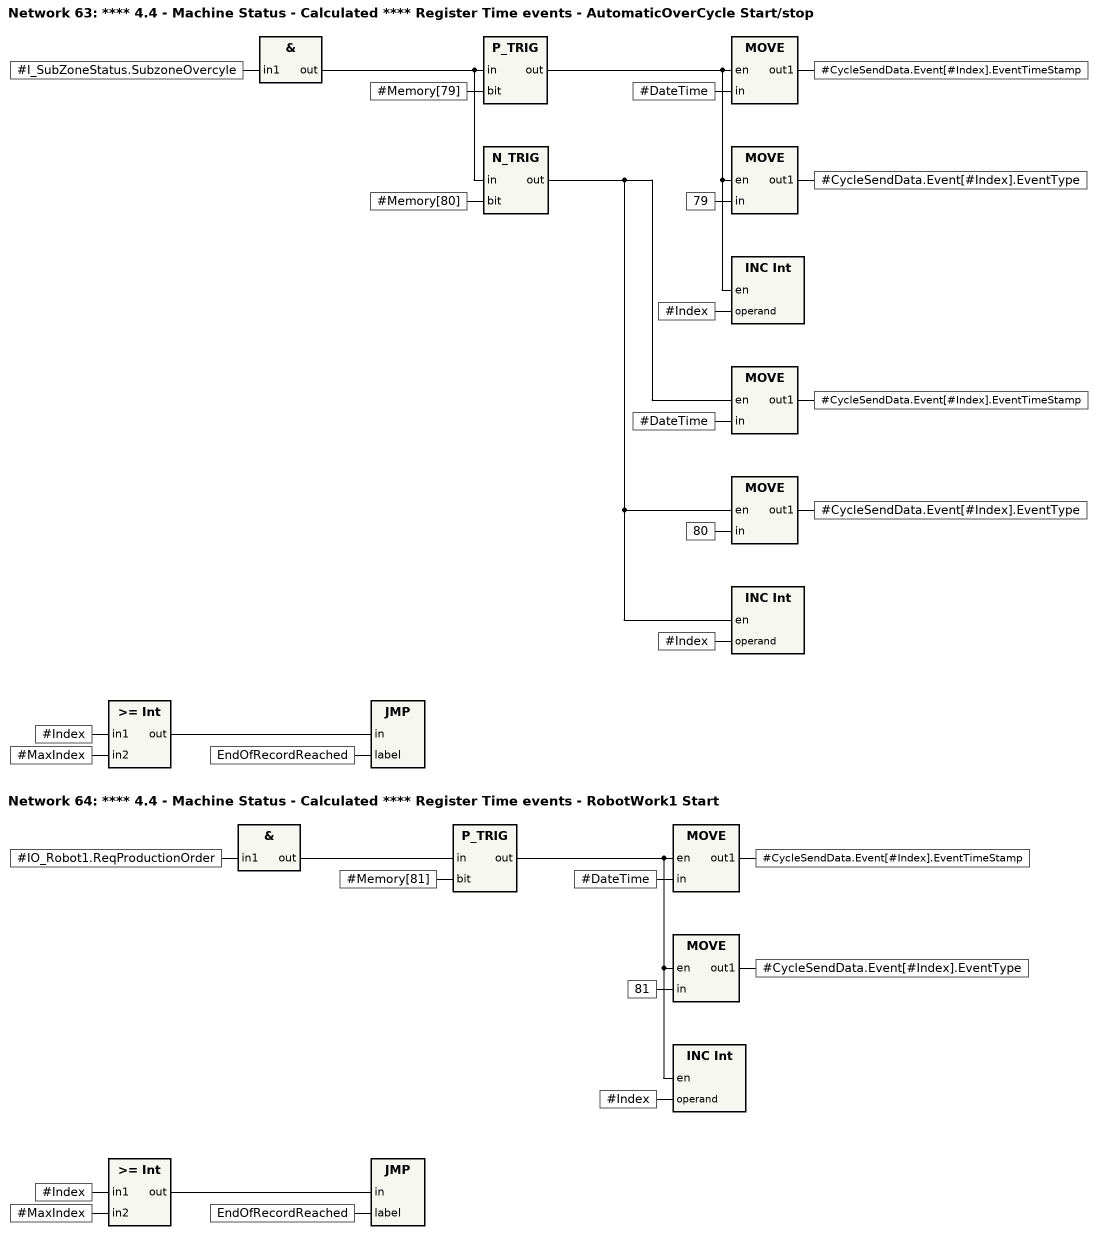
   #_w1 := #I_SubZoneStatus.SubzoneOvercyle AND NOT #Memory[79];   // rising edge
   #Memory[79] := #I_SubZoneStatus.SubzoneOvercyle;
   IF #_w1 THEN
       #CycleSendData.Event[#Index].EventTimeStamp := #DateTime;
       #CycleSendData.Event[#Index].EventType := 79;
       #Index := #Index + 1;
   END_IF;
   #_w2 := NOT #I_SubZoneStatus.SubzoneOvercyle AND #Memory[80];   // falling edge
   #Memory[80] := #I_SubZoneStatus.SubzoneOvercyle;
   IF #_w2 THEN
       #CycleSendData.Event[#Index].EventTimeStamp := #DateTime;
       #CycleSendData.Event[#Index].EventType := 80;
       #Index := #Index + 1;
   END_IF;
   IF #Index >= #MaxIndex THEN GOTO EndOfRecordReached; END_IF;
END_REGION

REGION Network 64: **** 4.4 - Machine Status - Calculated **** Register Time events - RobotWork1 Start
   #_w1 := #IO_Robot1.ReqProductionOrder AND NOT #Memory[81];   // rising edge
   #Memory[81] := #IO_Robot1.ReqProductionOrder;
   IF #_w1 THEN
       #CycleSendData.Event[#Index].EventTimeStamp := #DateTime;
       #CycleSendData.Event[#Index].EventType := 81;
       #Index := #Index + 1;
   END_IF;
   IF #Index >= #MaxIndex THEN GOTO EndOfRecordReached; END_IF;
END_REGION

REGION Network 65: **** 4.4 - Machine Status - Calculated **** Register Time events - RobotWork1 Stop
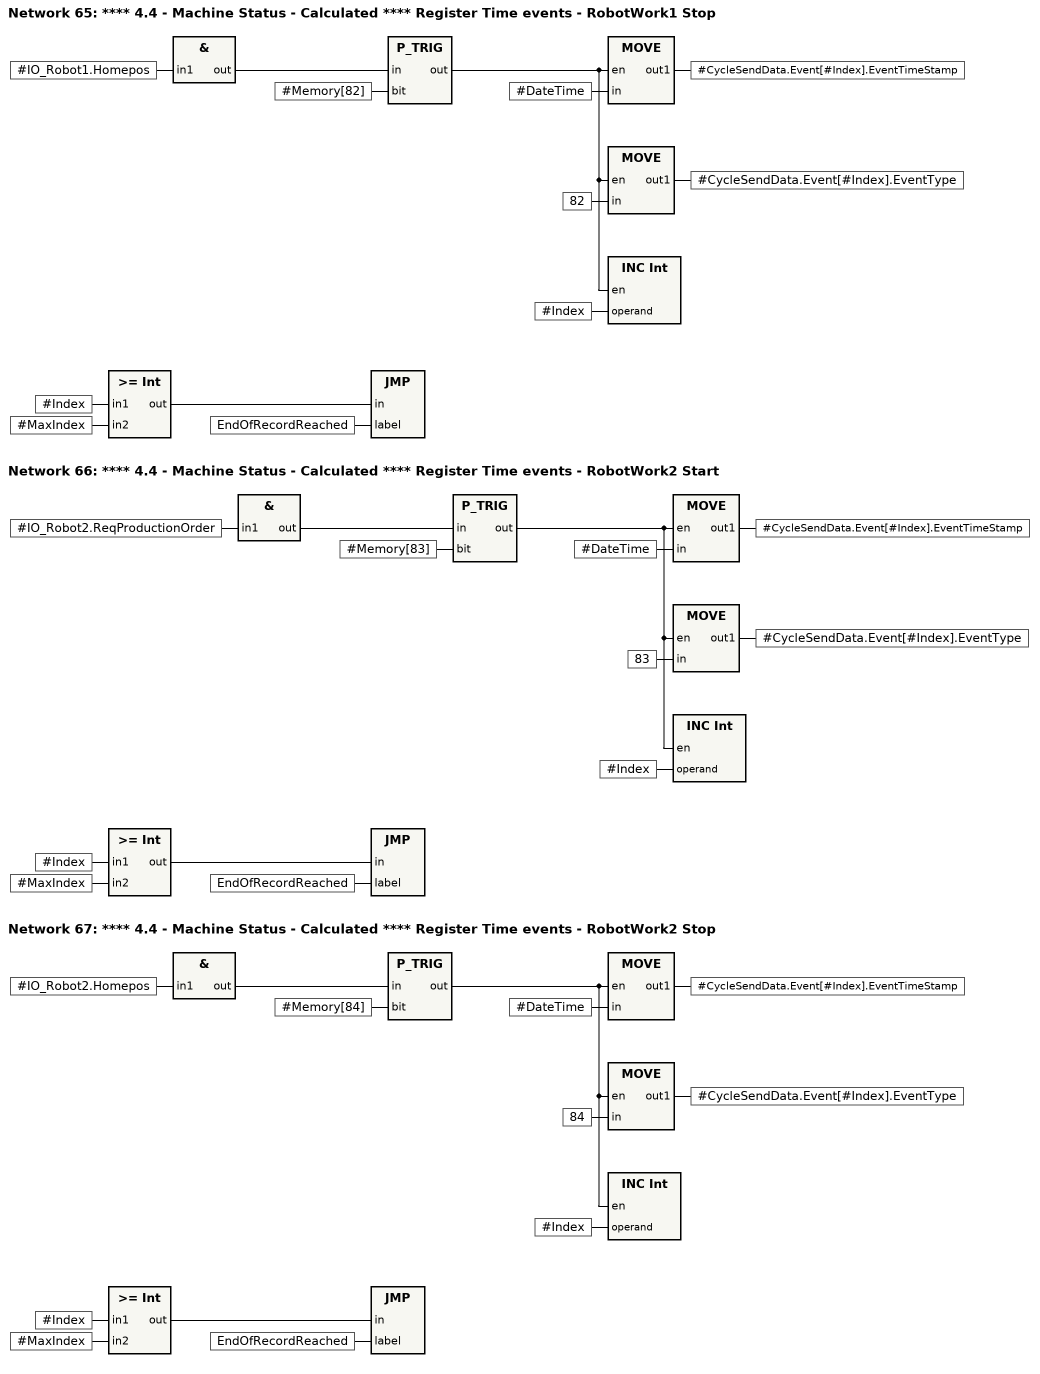
   #_w1 := #IO_Robot1.Homepos AND NOT #Memory[82];   // rising edge
   #Memory[82] := #IO_Robot1.Homepos;
   IF #_w1 THEN
       #CycleSendData.Event[#Index].EventTimeStamp := #DateTime;
       #CycleSendData.Event[#Index].EventType := 82;
       #Index := #Index + 1;
   END_IF;
   IF #Index >= #MaxIndex THEN GOTO EndOfRecordReached; END_IF;
END_REGION

REGION Network 66: **** 4.4 - Machine Status - Calculated **** Register Time events - RobotWork2 Start
   #_w1 := #IO_Robot2.ReqProductionOrder AND NOT #Memory[83];   // rising edge
   #Memory[83] := #IO_Robot2.ReqProductionOrder;
   IF #_w1 THEN
       #CycleSendData.Event[#Index].EventTimeStamp := #DateTime;
       #CycleSendData.Event[#Index].EventType := 83;
       #Index := #Index + 1;
   END_IF;
   IF #Index >= #MaxIndex THEN GOTO EndOfRecordReached; END_IF;
END_REGION

REGION Network 67: **** 4.4 - Machine Status - Calculated **** Register Time events - RobotWork2 Stop
   #_w1 := #IO_Robot2.Homepos AND NOT #Memory[84];   // rising edge
   #Memory[84] := #IO_Robot2.Homepos;
   IF #_w1 THEN
       #CycleSendData.Event[#Index].EventTimeStamp := #DateTime;
       #CycleSendData.Event[#Index].EventType := 84;
       #Index := #Index + 1;
   END_IF;
   IF #Index >= #MaxIndex THEN GOTO EndOfRecordReached; END_IF;
END_REGION

REGION Network 68: **** 4.4 - Machine Status - Calculated **** Register Time events - RobotWork3 Start
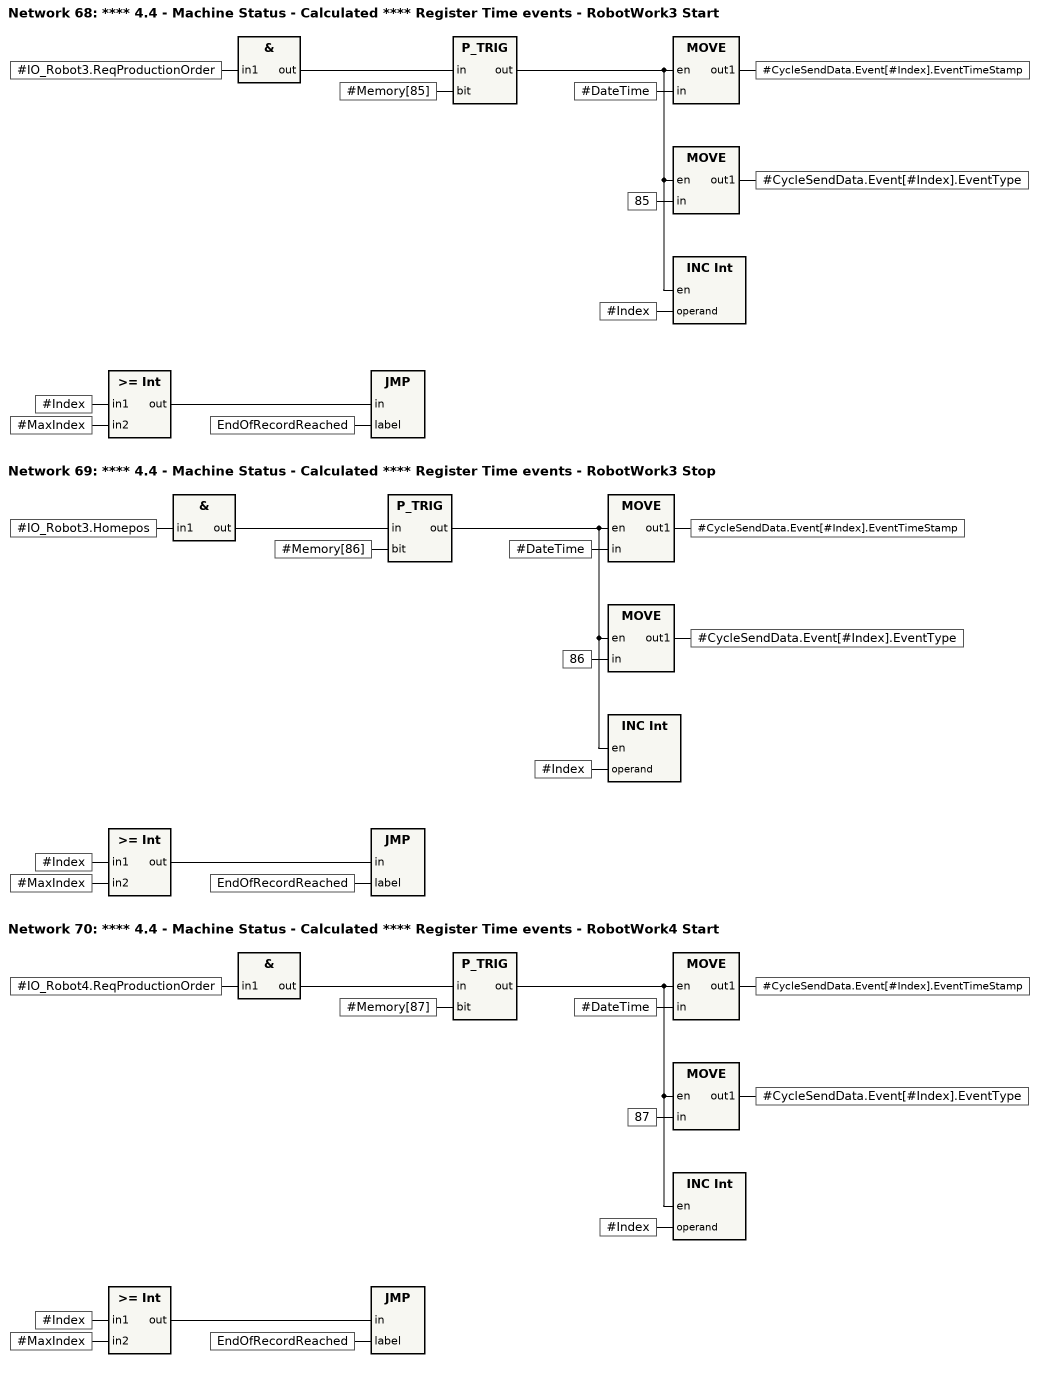
   #_w1 := #IO_Robot3.ReqProductionOrder AND NOT #Memory[85];   // rising edge
   #Memory[85] := #IO_Robot3.ReqProductionOrder;
   IF #_w1 THEN
       #CycleSendData.Event[#Index].EventTimeStamp := #DateTime;
       #CycleSendData.Event[#Index].EventType := 85;
       #Index := #Index + 1;
   END_IF;
   IF #Index >= #MaxIndex THEN GOTO EndOfRecordReached; END_IF;
END_REGION

REGION Network 69: **** 4.4 - Machine Status - Calculated **** Register Time events - RobotWork3 Stop
   #_w1 := #IO_Robot3.Homepos AND NOT #Memory[86];   // rising edge
   #Memory[86] := #IO_Robot3.Homepos;
   IF #_w1 THEN
       #CycleSendData.Event[#Index].EventTimeStamp := #DateTime;
       #CycleSendData.Event[#Index].EventType := 86;
       #Index := #Index + 1;
   END_IF;
   IF #Index >= #MaxIndex THEN GOTO EndOfRecordReached; END_IF;
END_REGION

REGION Network 70: **** 4.4 - Machine Status - Calculated **** Register Time events - RobotWork4 Start
   #_w1 := #IO_Robot4.ReqProductionOrder AND NOT #Memory[87];   // rising edge
   #Memory[87] := #IO_Robot4.ReqProductionOrder;
   IF #_w1 THEN
       #CycleSendData.Event[#Index].EventTimeStamp := #DateTime;
       #CycleSendData.Event[#Index].EventType := 87;
       #Index := #Index + 1;
   END_IF;
   IF #Index >= #MaxIndex THEN GOTO EndOfRecordReached; END_IF;
END_REGION

REGION Network 71: **** 4.4 - Machine Status - Calculated **** Register Time events - RobotWork4 Stop
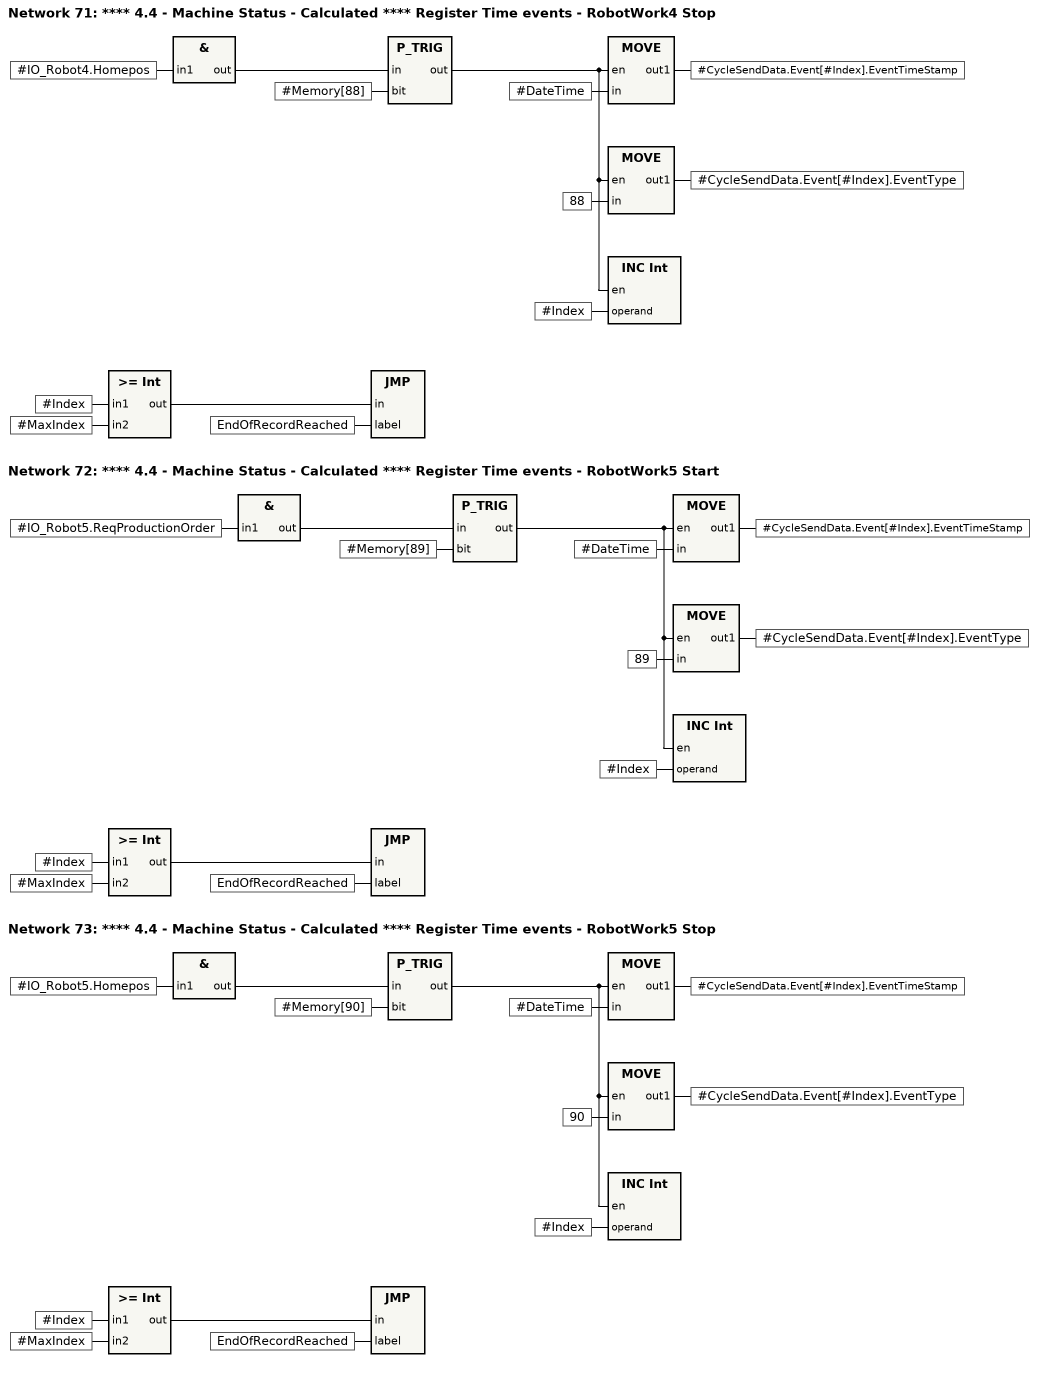
   #_w1 := #IO_Robot4.Homepos AND NOT #Memory[88];   // rising edge
   #Memory[88] := #IO_Robot4.Homepos;
   IF #_w1 THEN
       #CycleSendData.Event[#Index].EventTimeStamp := #DateTime;
       #CycleSendData.Event[#Index].EventType := 88;
       #Index := #Index + 1;
   END_IF;
   IF #Index >= #MaxIndex THEN GOTO EndOfRecordReached; END_IF;
END_REGION

REGION Network 72: **** 4.4 - Machine Status - Calculated **** Register Time events - RobotWork5 Start
   #_w1 := #IO_Robot5.ReqProductionOrder AND NOT #Memory[89];   // rising edge
   #Memory[89] := #IO_Robot5.ReqProductionOrder;
   IF #_w1 THEN
       #CycleSendData.Event[#Index].EventTimeStamp := #DateTime;
       #CycleSendData.Event[#Index].EventType := 89;
       #Index := #Index + 1;
   END_IF;
   IF #Index >= #MaxIndex THEN GOTO EndOfRecordReached; END_IF;
END_REGION

REGION Network 73: **** 4.4 - Machine Status - Calculated **** Register Time events - RobotWork5 Stop
   #_w1 := #IO_Robot5.Homepos AND NOT #Memory[90];   // rising edge
   #Memory[90] := #IO_Robot5.Homepos;
   IF #_w1 THEN
       #CycleSendData.Event[#Index].EventTimeStamp := #DateTime;
       #CycleSendData.Event[#Index].EventType := 90;
       #Index := #Index + 1;
   END_IF;
   IF #Index >= #MaxIndex THEN GOTO EndOfRecordReached; END_IF;
END_REGION

REGION Network 74: **** 4.4 - Machine Status - Calculated **** Register Time events - RobotWork6 Start
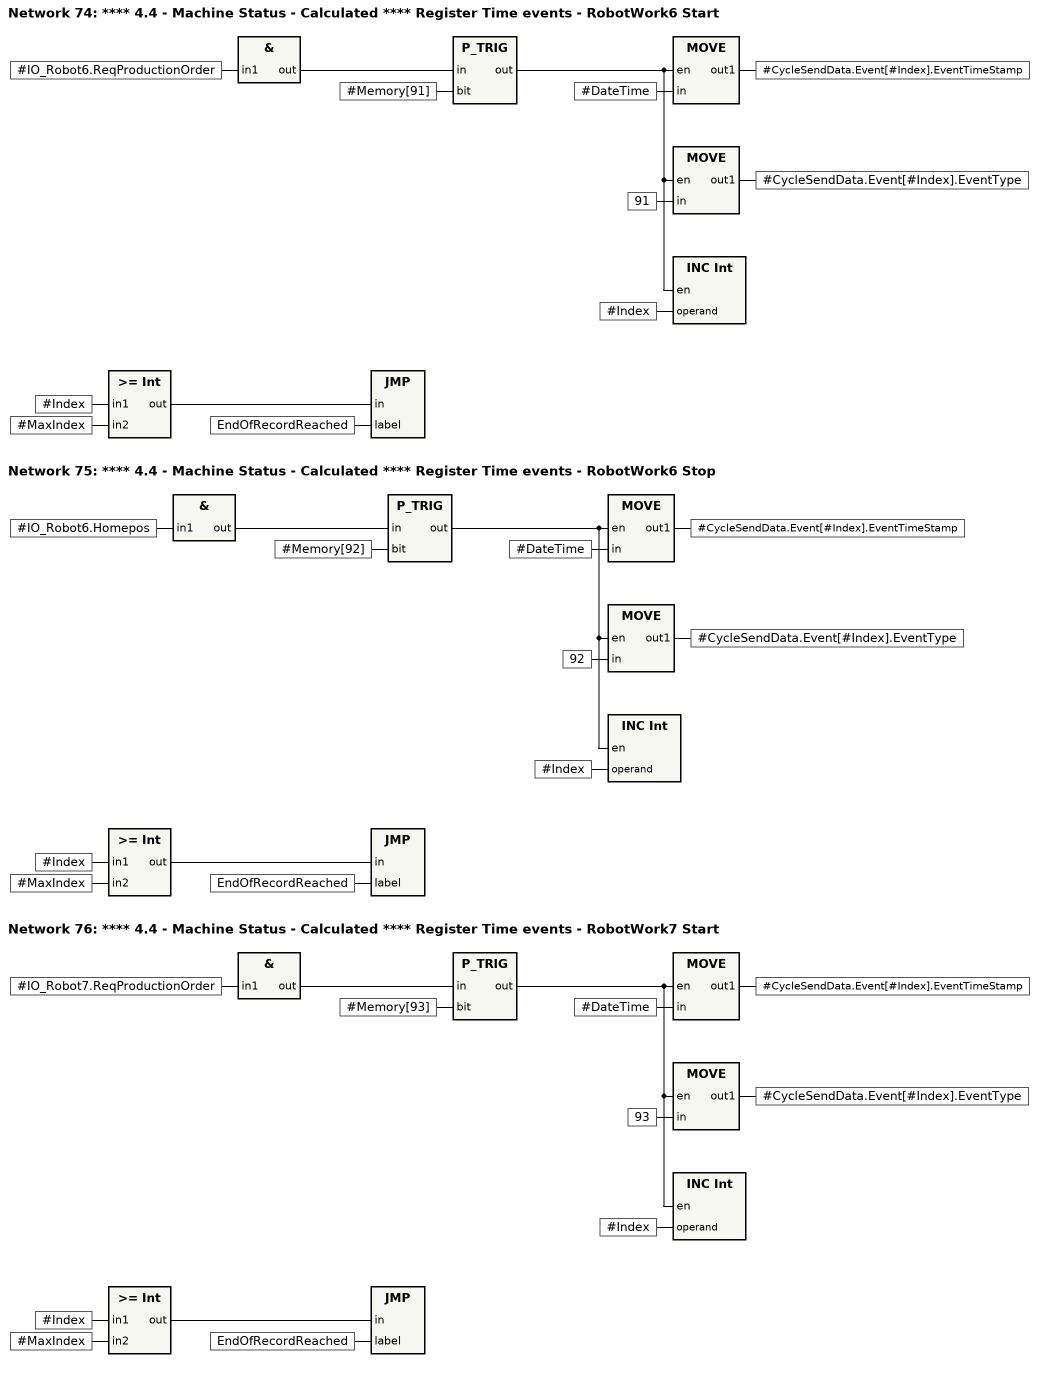
   #_w1 := #IO_Robot6.ReqProductionOrder AND NOT #Memory[91];   // rising edge
   #Memory[91] := #IO_Robot6.ReqProductionOrder;
   IF #_w1 THEN
       #CycleSendData.Event[#Index].EventTimeStamp := #DateTime;
       #CycleSendData.Event[#Index].EventType := 91;
       #Index := #Index + 1;
   END_IF;
   IF #Index >= #MaxIndex THEN GOTO EndOfRecordReached; END_IF;
END_REGION

REGION Network 75: **** 4.4 - Machine Status - Calculated **** Register Time events - RobotWork6 Stop
   #_w1 := #IO_Robot6.Homepos AND NOT #Memory[92];   // rising edge
   #Memory[92] := #IO_Robot6.Homepos;
   IF #_w1 THEN
       #CycleSendData.Event[#Index].EventTimeStamp := #DateTime;
       #CycleSendData.Event[#Index].EventType := 92;
       #Index := #Index + 1;
   END_IF;
   IF #Index >= #MaxIndex THEN GOTO EndOfRecordReached; END_IF;
END_REGION

REGION Network 76: **** 4.4 - Machine Status - Calculated **** Register Time events - RobotWork7 Start
   #_w1 := #IO_Robot7.ReqProductionOrder AND NOT #Memory[93];   // rising edge
   #Memory[93] := #IO_Robot7.ReqProductionOrder;
   IF #_w1 THEN
       #CycleSendData.Event[#Index].EventTimeStamp := #DateTime;
       #CycleSendData.Event[#Index].EventType := 93;
       #Index := #Index + 1;
   END_IF;
   IF #Index >= #MaxIndex THEN GOTO EndOfRecordReached; END_IF;
END_REGION

REGION Network 77: **** 4.4 - Machine Status - Calculated **** Register Time events - RobotWork7 Stop
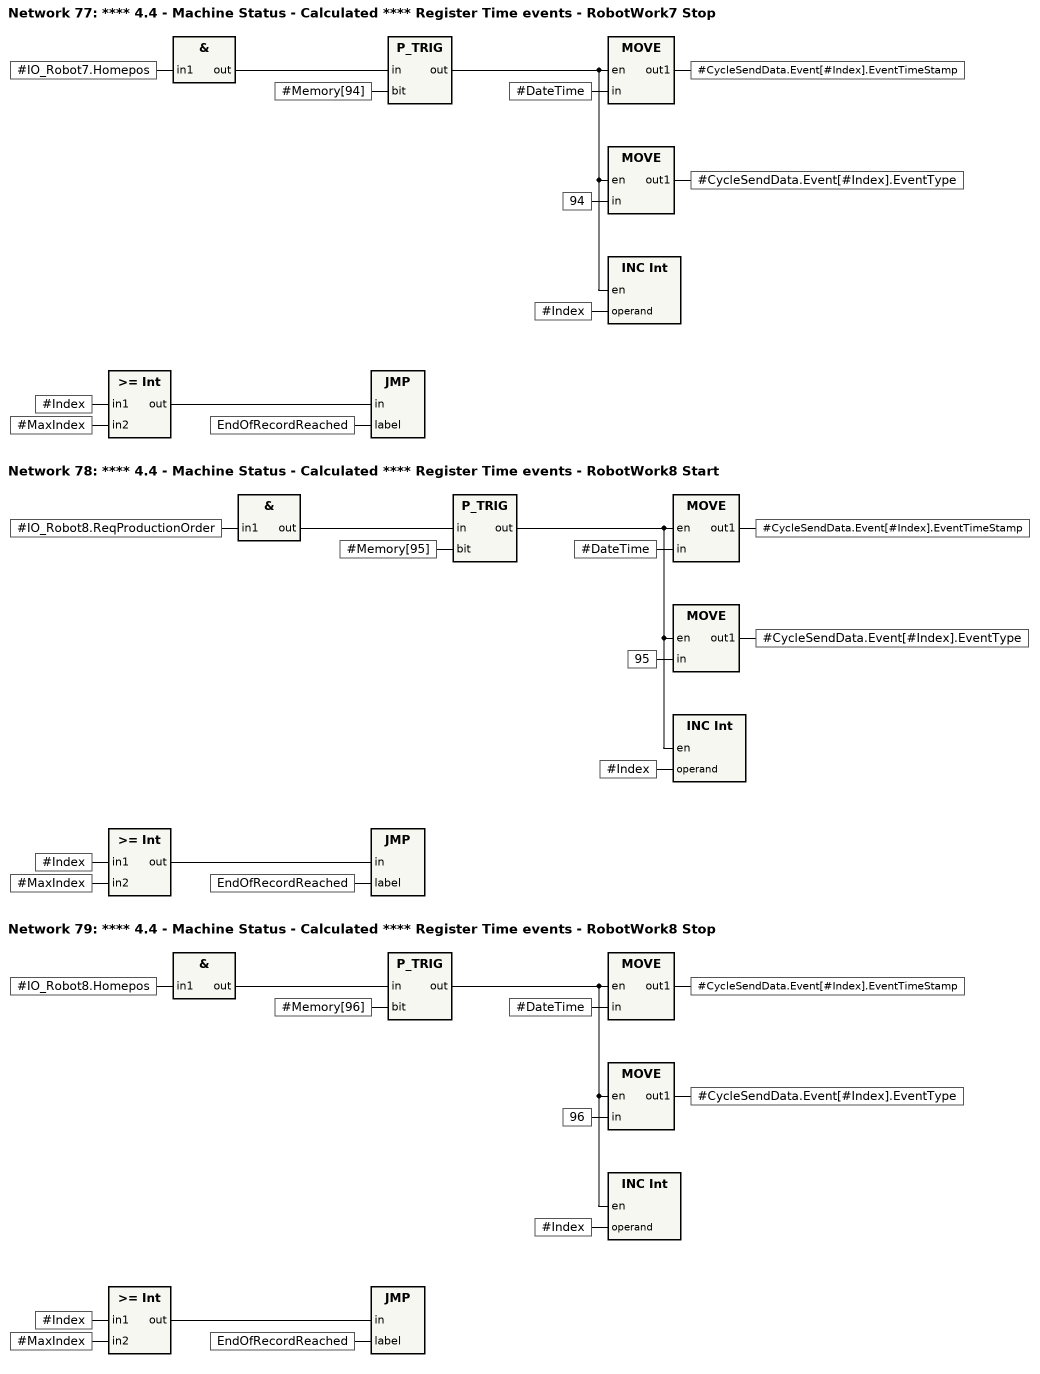
   #_w1 := #IO_Robot7.Homepos AND NOT #Memory[94];   // rising edge
   #Memory[94] := #IO_Robot7.Homepos;
   IF #_w1 THEN
       #CycleSendData.Event[#Index].EventTimeStamp := #DateTime;
       #CycleSendData.Event[#Index].EventType := 94;
       #Index := #Index + 1;
   END_IF;
   IF #Index >= #MaxIndex THEN GOTO EndOfRecordReached; END_IF;
END_REGION

REGION Network 78: **** 4.4 - Machine Status - Calculated **** Register Time events - RobotWork8 Start
   #_w1 := #IO_Robot8.ReqProductionOrder AND NOT #Memory[95];   // rising edge
   #Memory[95] := #IO_Robot8.ReqProductionOrder;
   IF #_w1 THEN
       #CycleSendData.Event[#Index].EventTimeStamp := #DateTime;
       #CycleSendData.Event[#Index].EventType := 95;
       #Index := #Index + 1;
   END_IF;
   IF #Index >= #MaxIndex THEN GOTO EndOfRecordReached; END_IF;
END_REGION

REGION Network 79: **** 4.4 - Machine Status - Calculated **** Register Time events - RobotWork8 Stop
   #_w1 := #IO_Robot8.Homepos AND NOT #Memory[96];   // rising edge
   #Memory[96] := #IO_Robot8.Homepos;
   IF #_w1 THEN
       #CycleSendData.Event[#Index].EventTimeStamp := #DateTime;
       #CycleSendData.Event[#Index].EventType := 96;
       #Index := #Index + 1;
   END_IF;
   IF #Index >= #MaxIndex THEN GOTO EndOfRecordReached; END_IF;
END_REGION

REGION Network 80: **** 4.4 - Machine Status - Calculated **** Register Time events - RobotWork9 Start
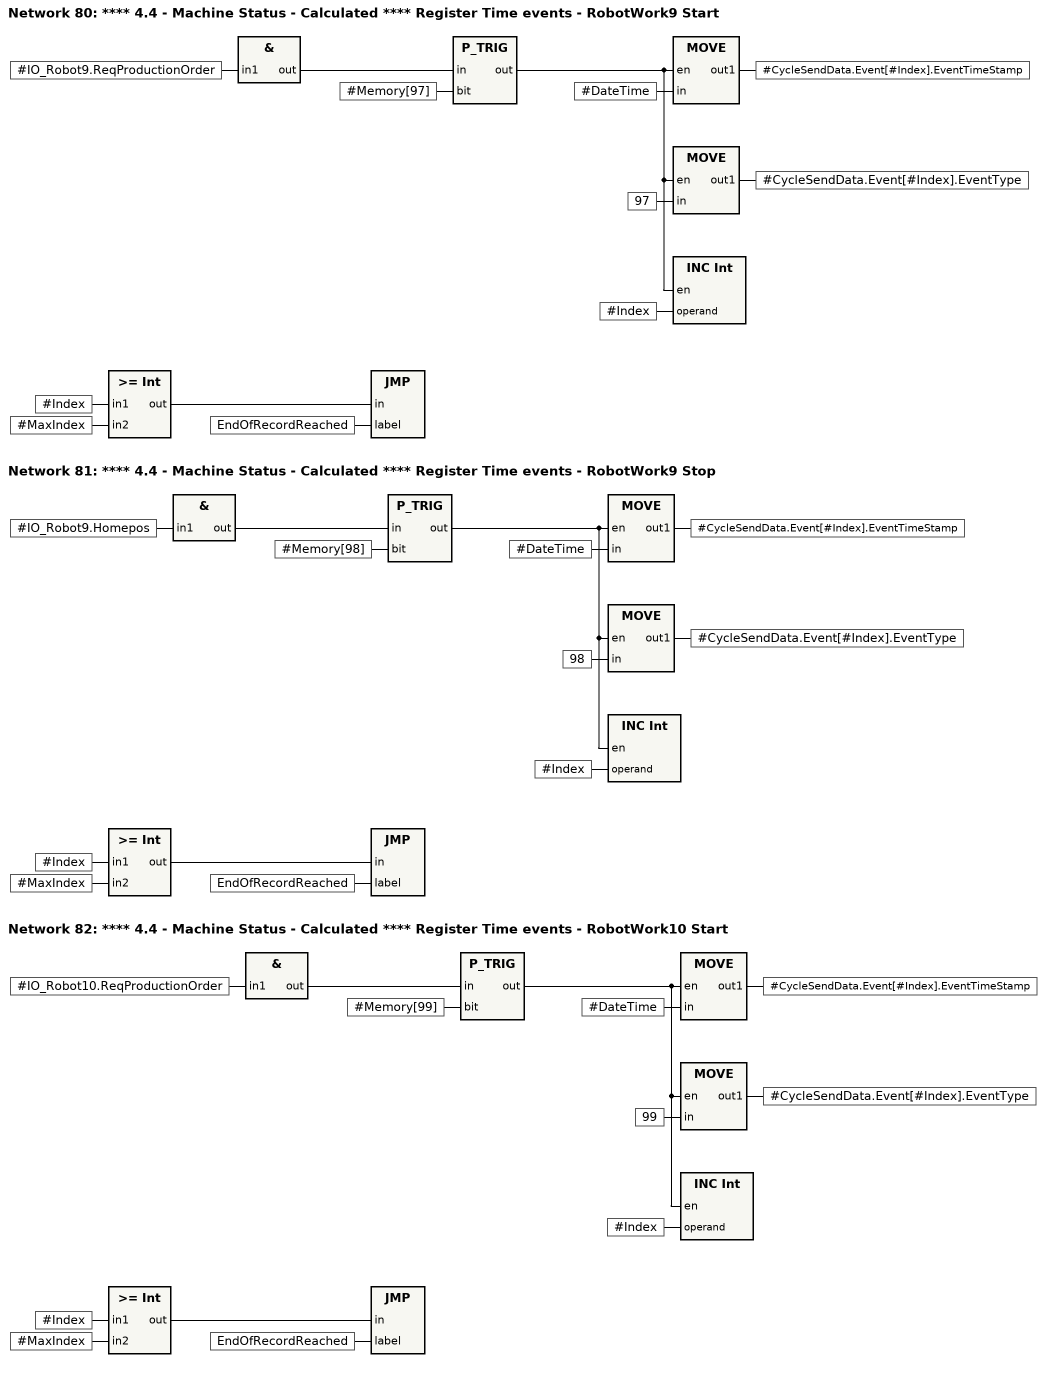
   #_w1 := #IO_Robot9.ReqProductionOrder AND NOT #Memory[97];   // rising edge
   #Memory[97] := #IO_Robot9.ReqProductionOrder;
   IF #_w1 THEN
       #CycleSendData.Event[#Index].EventTimeStamp := #DateTime;
       #CycleSendData.Event[#Index].EventType := 97;
       #Index := #Index + 1;
   END_IF;
   IF #Index >= #MaxIndex THEN GOTO EndOfRecordReached; END_IF;
END_REGION

REGION Network 81: **** 4.4 - Machine Status - Calculated **** Register Time events - RobotWork9 Stop
   #_w1 := #IO_Robot9.Homepos AND NOT #Memory[98];   // rising edge
   #Memory[98] := #IO_Robot9.Homepos;
   IF #_w1 THEN
       #CycleSendData.Event[#Index].EventTimeStamp := #DateTime;
       #CycleSendData.Event[#Index].EventType := 98;
       #Index := #Index + 1;
   END_IF;
   IF #Index >= #MaxIndex THEN GOTO EndOfRecordReached; END_IF;
END_REGION

REGION Network 82: **** 4.4 - Machine Status - Calculated **** Register Time events - RobotWork10 Start
   #_w1 := #IO_Robot10.ReqProductionOrder AND NOT #Memory[99];   // rising edge
   #Memory[99] := #IO_Robot10.ReqProductionOrder;
   IF #_w1 THEN
       #CycleSendData.Event[#Index].EventTimeStamp := #DateTime;
       #CycleSendData.Event[#Index].EventType := 99;
       #Index := #Index + 1;
   END_IF;
   IF #Index >= #MaxIndex THEN GOTO EndOfRecordReached; END_IF;
END_REGION

REGION Network 83: **** 4.4 - Machine Status - Calculated **** Register Time events - RobotWork10 Stop
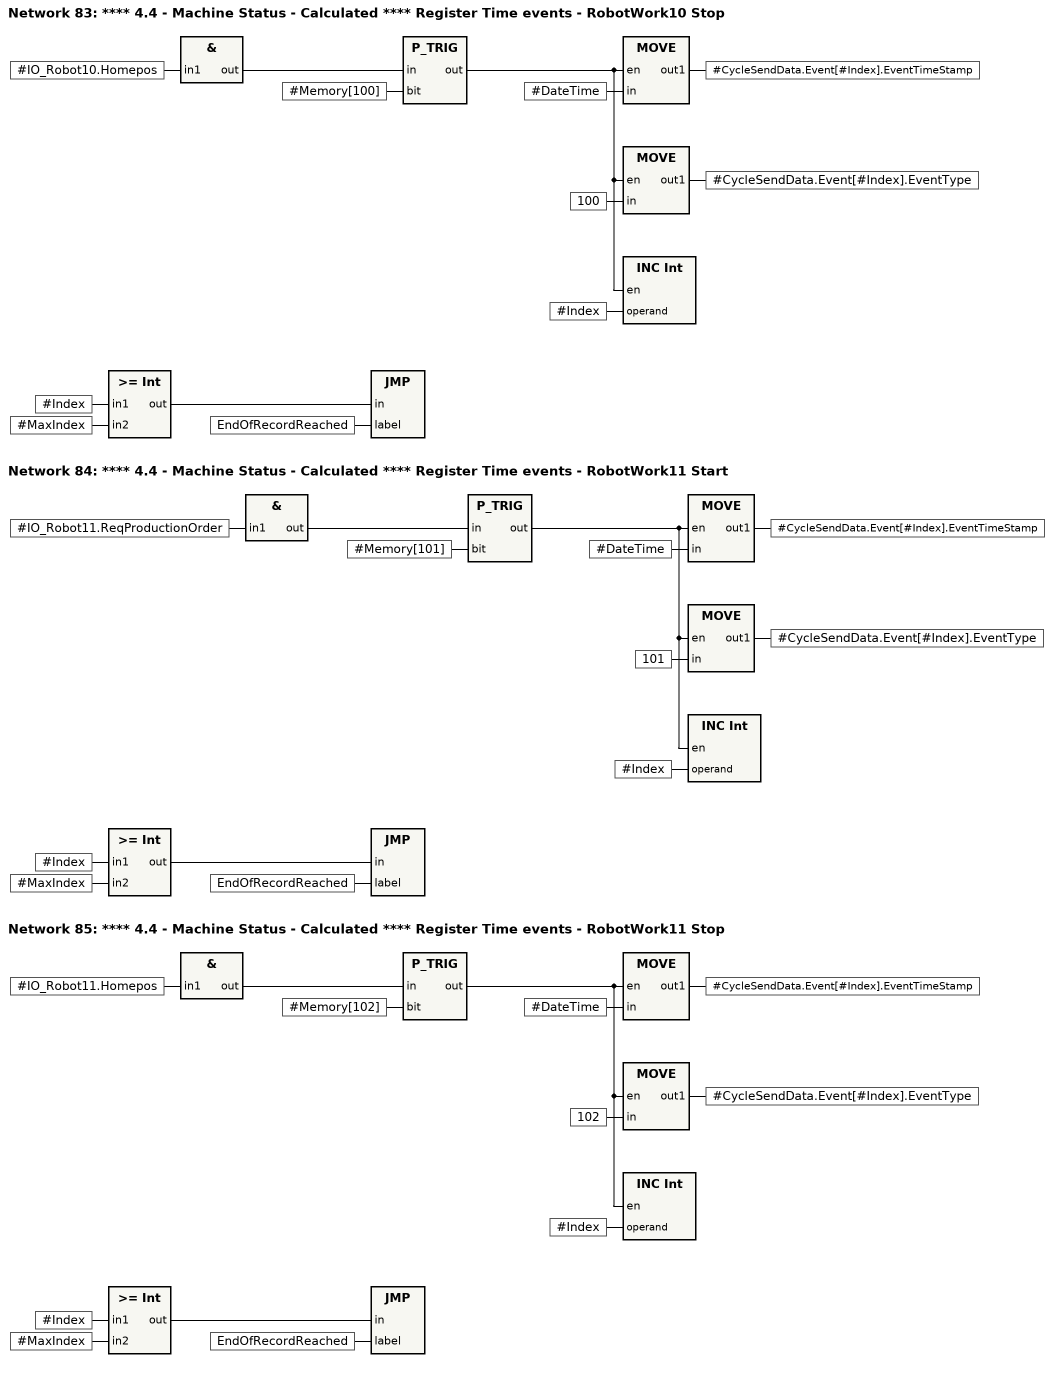
   #_w1 := #IO_Robot10.Homepos AND NOT #Memory[100];   // rising edge
   #Memory[100] := #IO_Robot10.Homepos;
   IF #_w1 THEN
       #CycleSendData.Event[#Index].EventTimeStamp := #DateTime;
       #CycleSendData.Event[#Index].EventType := 100;
       #Index := #Index + 1;
   END_IF;
   IF #Index >= #MaxIndex THEN GOTO EndOfRecordReached; END_IF;
END_REGION

REGION Network 84: **** 4.4 - Machine Status - Calculated **** Register Time events - RobotWork11 Start
   #_w1 := #IO_Robot11.ReqProductionOrder AND NOT #Memory[101];   // rising edge
   #Memory[101] := #IO_Robot11.ReqProductionOrder;
   IF #_w1 THEN
       #CycleSendData.Event[#Index].EventTimeStamp := #DateTime;
       #CycleSendData.Event[#Index].EventType := 101;
       #Index := #Index + 1;
   END_IF;
   IF #Index >= #MaxIndex THEN GOTO EndOfRecordReached; END_IF;
END_REGION

REGION Network 85: **** 4.4 - Machine Status - Calculated **** Register Time events - RobotWork11 Stop
   #_w1 := #IO_Robot11.Homepos AND NOT #Memory[102];   // rising edge
   #Memory[102] := #IO_Robot11.Homepos;
   IF #_w1 THEN
       #CycleSendData.Event[#Index].EventTimeStamp := #DateTime;
       #CycleSendData.Event[#Index].EventType := 102;
       #Index := #Index + 1;
   END_IF;
   IF #Index >= #MaxIndex THEN GOTO EndOfRecordReached; END_IF;
END_REGION

REGION Network 86: **** 4.4 - Machine Status - Calculated **** Register Time events - RobotWork12 Start
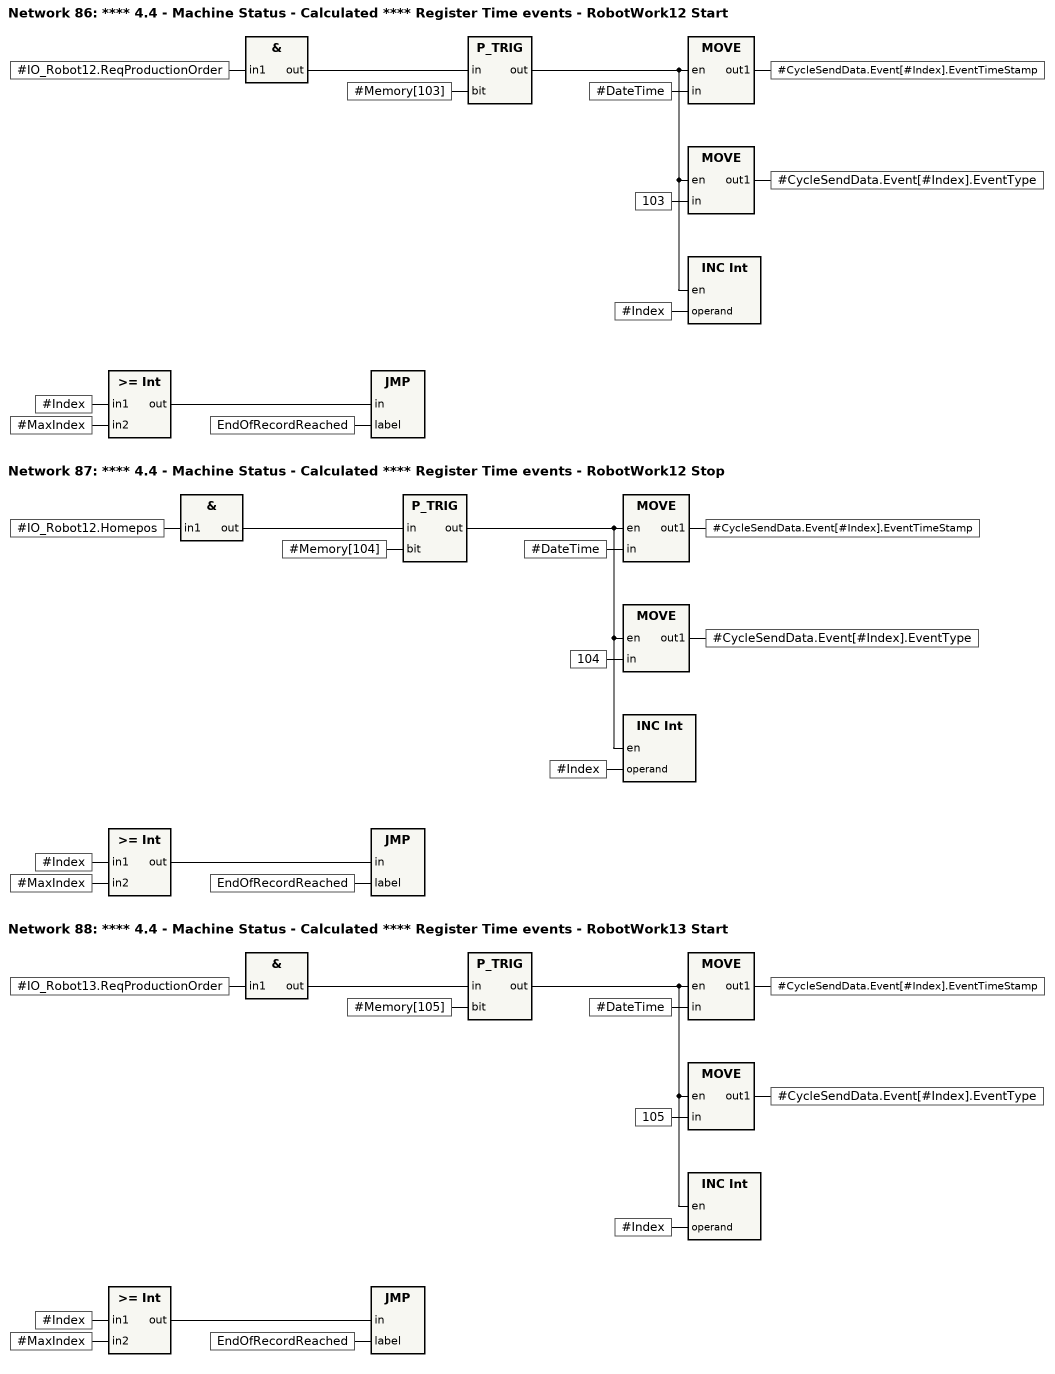
   #_w1 := #IO_Robot12.ReqProductionOrder AND NOT #Memory[103];   // rising edge
   #Memory[103] := #IO_Robot12.ReqProductionOrder;
   IF #_w1 THEN
       #CycleSendData.Event[#Index].EventTimeStamp := #DateTime;
       #CycleSendData.Event[#Index].EventType := 103;
       #Index := #Index + 1;
   END_IF;
   IF #Index >= #MaxIndex THEN GOTO EndOfRecordReached; END_IF;
END_REGION

REGION Network 87: **** 4.4 - Machine Status - Calculated **** Register Time events - RobotWork12 Stop
   #_w1 := #IO_Robot12.Homepos AND NOT #Memory[104];   // rising edge
   #Memory[104] := #IO_Robot12.Homepos;
   IF #_w1 THEN
       #CycleSendData.Event[#Index].EventTimeStamp := #DateTime;
       #CycleSendData.Event[#Index].EventType := 104;
       #Index := #Index + 1;
   END_IF;
   IF #Index >= #MaxIndex THEN GOTO EndOfRecordReached; END_IF;
END_REGION

REGION Network 88: **** 4.4 - Machine Status - Calculated **** Register Time events - RobotWork13 Start
   #_w1 := #IO_Robot13.ReqProductionOrder AND NOT #Memory[105];   // rising edge
   #Memory[105] := #IO_Robot13.ReqProductionOrder;
   IF #_w1 THEN
       #CycleSendData.Event[#Index].EventTimeStamp := #DateTime;
       #CycleSendData.Event[#Index].EventType := 105;
       #Index := #Index + 1;
   END_IF;
   IF #Index >= #MaxIndex THEN GOTO EndOfRecordReached; END_IF;
END_REGION

REGION Network 89: **** 4.4 - Machine Status - Calculated **** Register Time events - RobotWork13 Stop
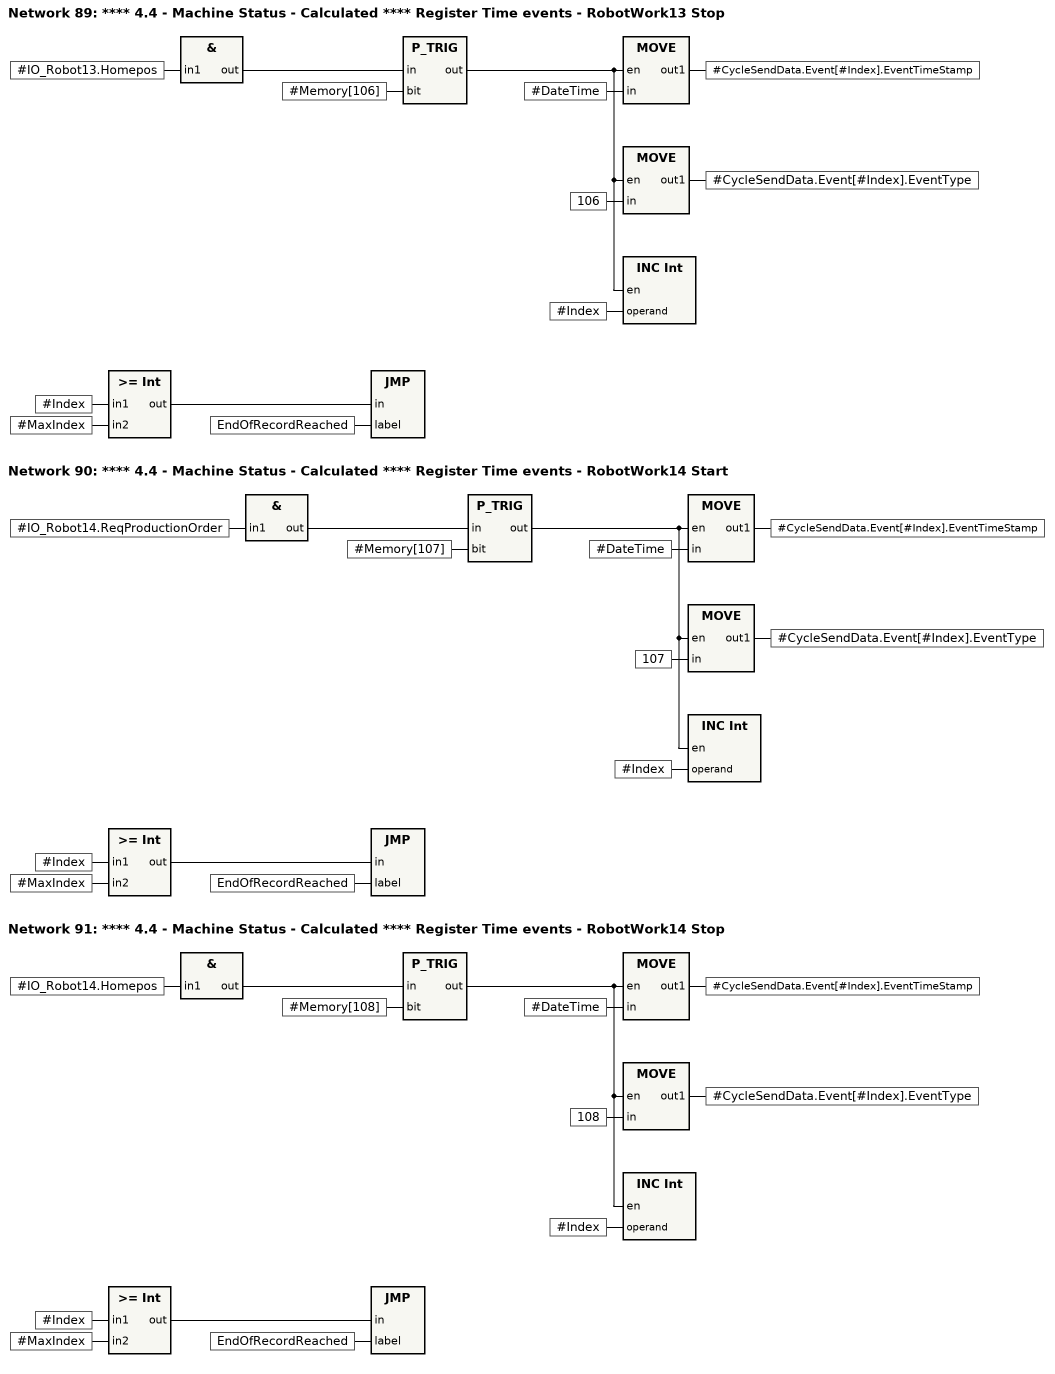
   #_w1 := #IO_Robot13.Homepos AND NOT #Memory[106];   // rising edge
   #Memory[106] := #IO_Robot13.Homepos;
   IF #_w1 THEN
       #CycleSendData.Event[#Index].EventTimeStamp := #DateTime;
       #CycleSendData.Event[#Index].EventType := 106;
       #Index := #Index + 1;
   END_IF;
   IF #Index >= #MaxIndex THEN GOTO EndOfRecordReached; END_IF;
END_REGION

REGION Network 90: **** 4.4 - Machine Status - Calculated **** Register Time events - RobotWork14 Start
   #_w1 := #IO_Robot14.ReqProductionOrder AND NOT #Memory[107];   // rising edge
   #Memory[107] := #IO_Robot14.ReqProductionOrder;
   IF #_w1 THEN
       #CycleSendData.Event[#Index].EventTimeStamp := #DateTime;
       #CycleSendData.Event[#Index].EventType := 107;
       #Index := #Index + 1;
   END_IF;
   IF #Index >= #MaxIndex THEN GOTO EndOfRecordReached; END_IF;
END_REGION

REGION Network 91: **** 4.4 - Machine Status - Calculated **** Register Time events - RobotWork14 Stop
   #_w1 := #IO_Robot14.Homepos AND NOT #Memory[108];   // rising edge
   #Memory[108] := #IO_Robot14.Homepos;
   IF #_w1 THEN
       #CycleSendData.Event[#Index].EventTimeStamp := #DateTime;
       #CycleSendData.Event[#Index].EventType := 108;
       #Index := #Index + 1;
   END_IF;
   IF #Index >= #MaxIndex THEN GOTO EndOfRecordReached; END_IF;
END_REGION

REGION Network 92: **** 4.4 - Machine Status - Calculated **** Register Time events - ProcessCycle Stop - EndOfRecordReached LABEL
   // Jump to this location in case the event record is full
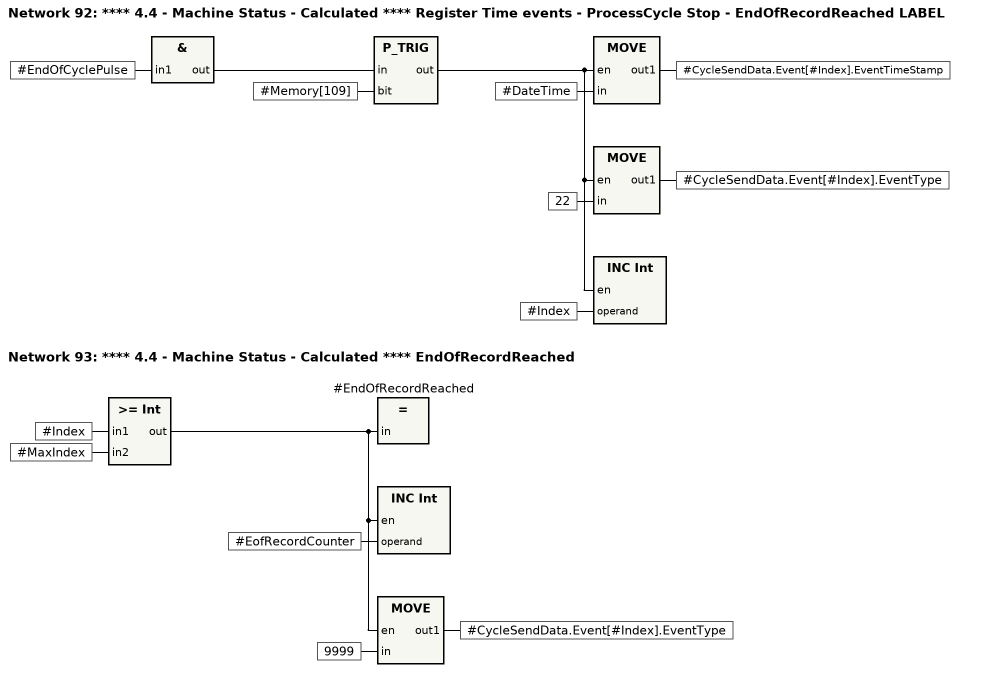
   EndOfRecordReached:
   #_w1 := #EndOfCyclePulse AND NOT #Memory[109];   // rising edge
   #Memory[109] := #EndOfCyclePulse;
   IF #_w1 THEN
       #CycleSendData.Event[#Index].EventTimeStamp := #DateTime;
       #CycleSendData.Event[#Index].EventType := 22;
       #Index := #Index + 1;
   END_IF;
END_REGION

REGION Network 93: **** 4.4 - Machine Status - Calculated **** EndOfRecordReached
   // When at end of record position, then count EofRecordCount AND mark enf of record event
   #EndOfRecordReached := #Index >= #MaxIndex;
   IF #EndOfRecordReached THEN
       #EofRecordCounter := #EofRecordCounter + 1;
       #CycleSendData.Event[#Index].EventType := 9999;
   END_IF;
END_REGION

REGION Network 94: **** 4.4 - Machine Status - Calculated **** At the End of cycle
   // Update figures at the end of the cycle
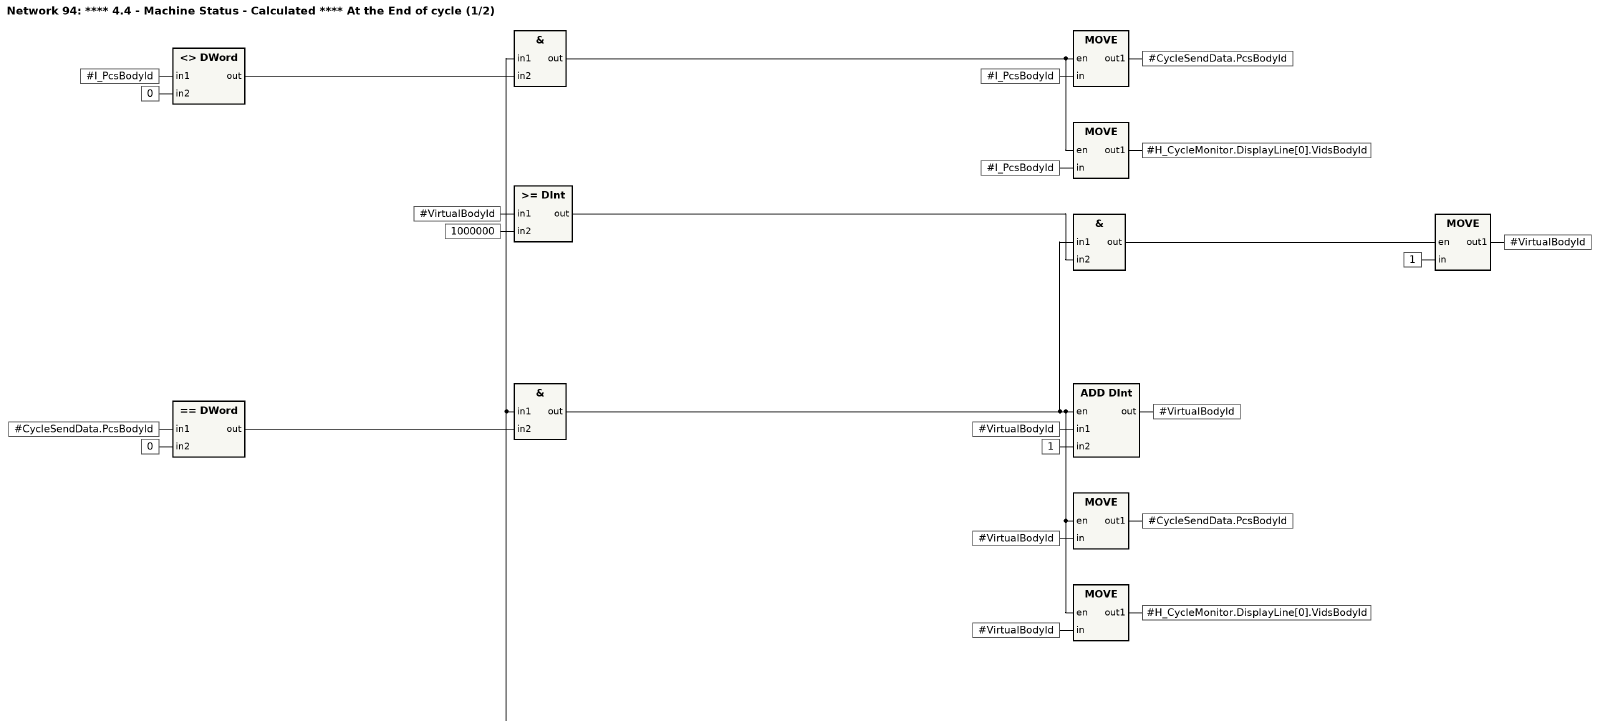
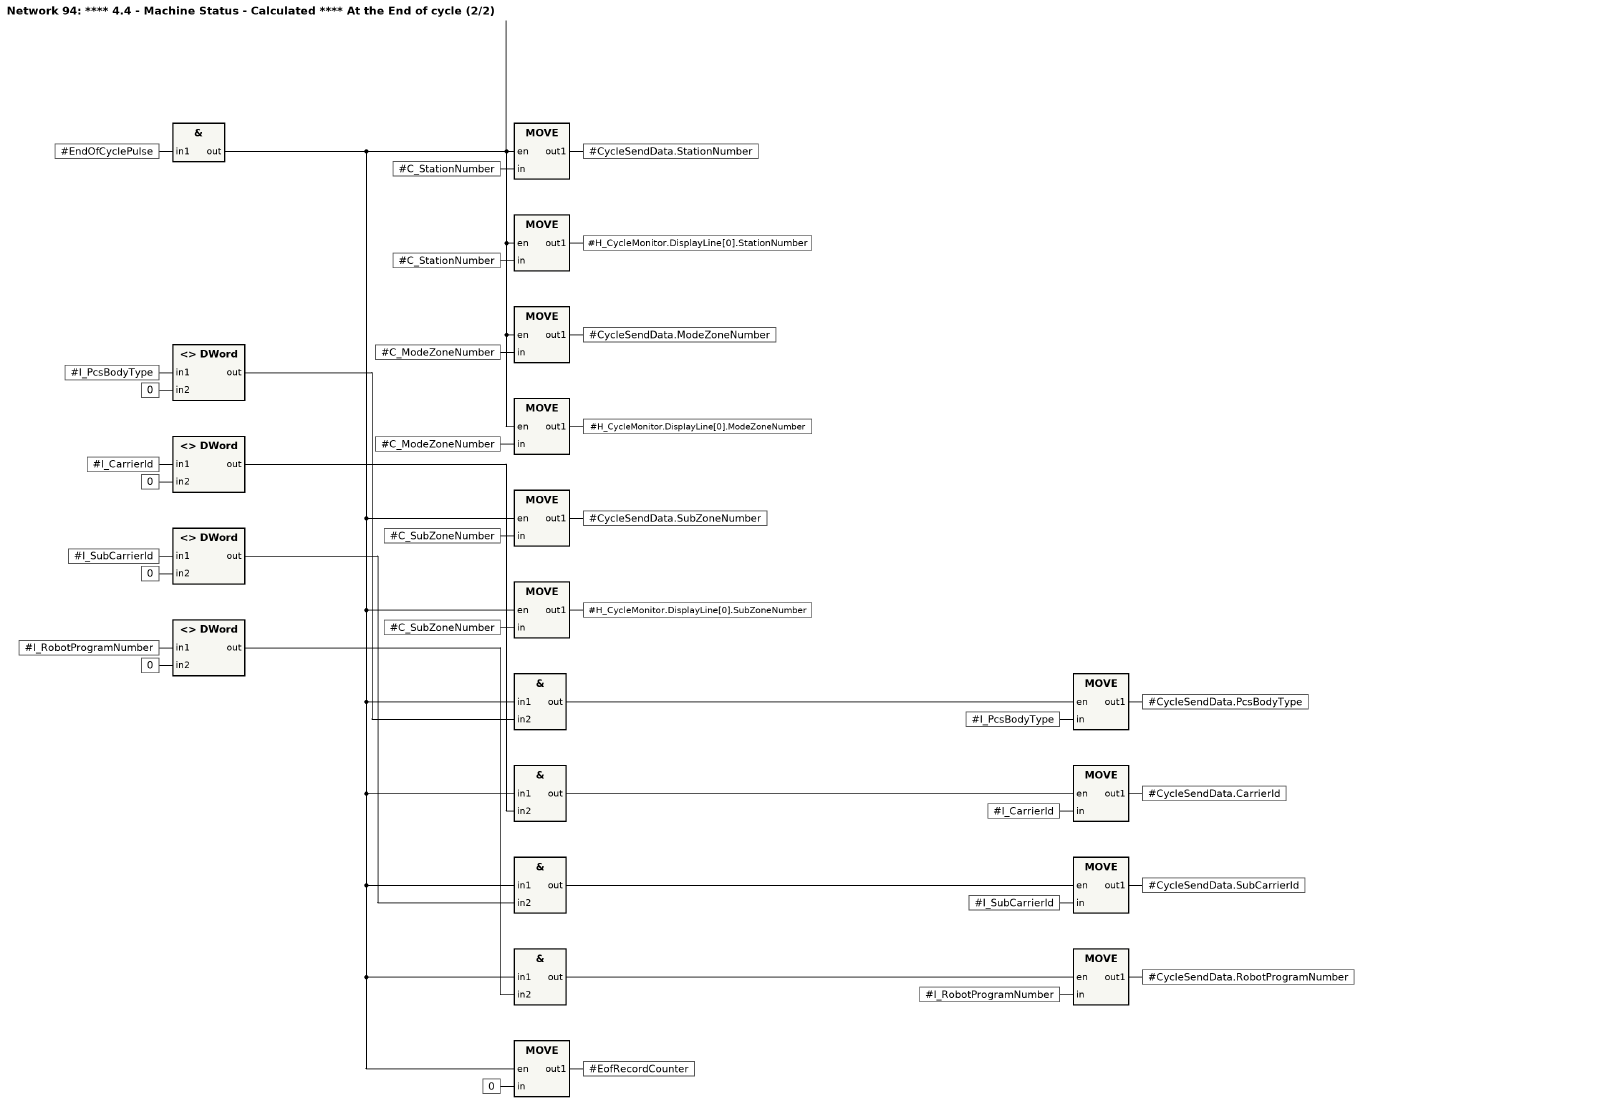
   IF #EndOfCyclePulse THEN
       #CycleSendData.StationNumber := #C_StationNumber;
       #H_CycleMonitor.DisplayLine[0].StationNumber := #C_StationNumber;
       #CycleSendData.ModeZoneNumber := #C_ModeZoneNumber;
       #H_CycleMonitor.DisplayLine[0].ModeZoneNumber := #C_ModeZoneNumber;
       #CycleSendData.SubZoneNumber := #C_SubZoneNumber;
       #H_CycleMonitor.DisplayLine[0].SubZoneNumber := #C_SubZoneNumber;
   END_IF;
   IF #EndOfCyclePulse AND (#I_PcsBodyId <> 0) THEN
       #CycleSendData.PcsBodyId := #I_PcsBodyId;
       #H_CycleMonitor.DisplayLine[0].VidsBodyId := #I_PcsBodyId;
   END_IF;
   #_w1 := #EndOfCyclePulse AND (#CycleSendData.PcsBodyId = 0);
   IF #_w1 THEN #VirtualBodyId := #VirtualBodyId + 1; END_IF;
   IF #_w1 AND (#VirtualBodyId >= 1000000) THEN #VirtualBodyId := 1; END_IF;
   IF #_w1 THEN
       #CycleSendData.PcsBodyId := #VirtualBodyId;
       #H_CycleMonitor.DisplayLine[0].VidsBodyId := #VirtualBodyId;
   END_IF;
   IF #EndOfCyclePulse AND (#I_PcsBodyType <> 0) THEN #CycleSendData.PcsBodyType := #I_PcsBodyType; END_IF;
   IF #EndOfCyclePulse AND (#I_CarrierId <> 0) THEN #CycleSendData.CarrierId := #I_CarrierId; END_IF;
   IF #EndOfCyclePulse AND (#I_SubCarrierId <> 0) THEN
       #CycleSendData.SubCarrierId := #I_SubCarrierId;
   END_IF;
   IF #EndOfCyclePulse AND (#I_RobotProgramNumber <> 0) THEN
       #CycleSendData.RobotProgramNumber := #I_RobotProgramNumber;
   END_IF;
   IF #EndOfCyclePulse THEN #EofRecordCounter := 0; END_IF;
END_REGION

REGION Network 95: **** 4.4 - Machine Status - Calculated **** Store Accumulated times in first display line
   // Move data from local stack to first display line
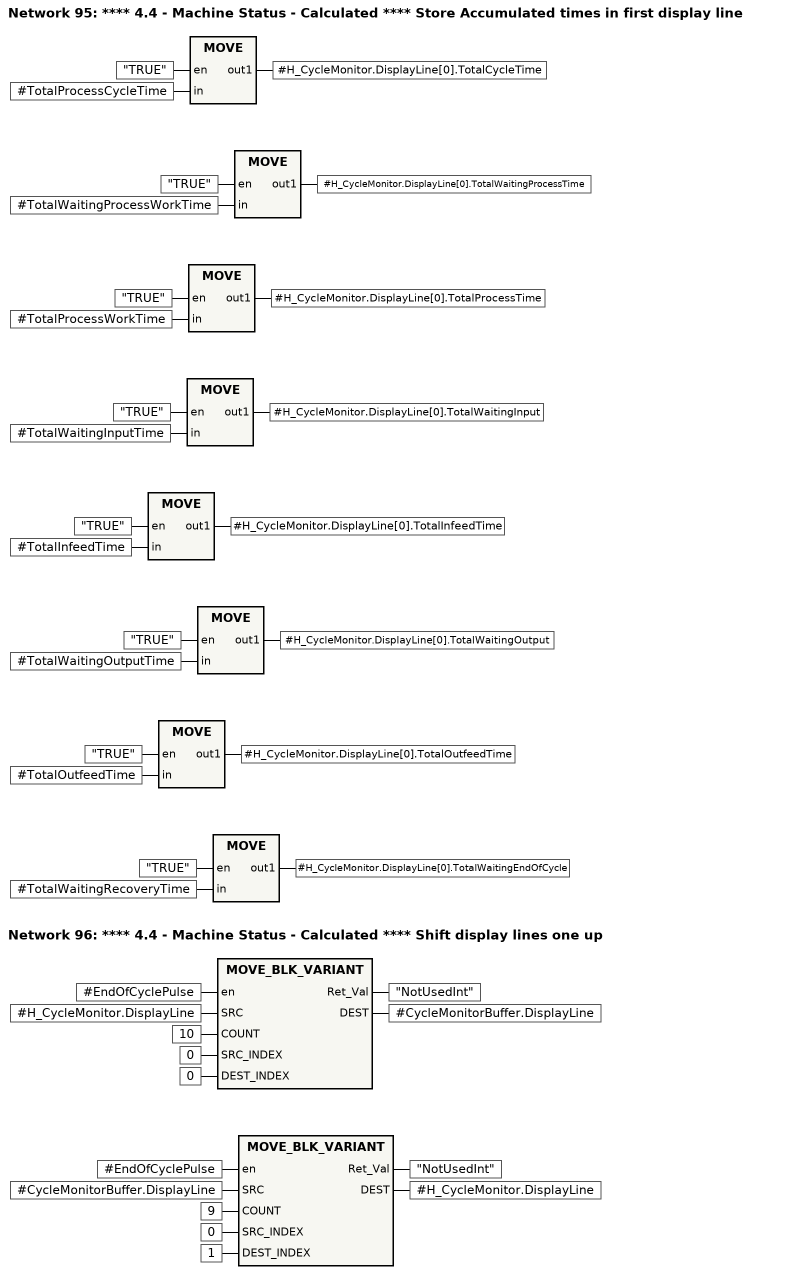
   IF "TRUE" THEN
       #H_CycleMonitor.DisplayLine[0].TotalCycleTime := #TotalProcessCycleTime;
       #H_CycleMonitor.DisplayLine[0].TotalWaitingProcessTime := #TotalWaitingProcessWorkTime;
       #H_CycleMonitor.DisplayLine[0].TotalProcessTime := #TotalProcessWorkTime;
       #H_CycleMonitor.DisplayLine[0].TotalWaitingInput := #TotalWaitingInputTime;
       #H_CycleMonitor.DisplayLine[0].TotalInfeedTime := #TotalInfeedTime;
       #H_CycleMonitor.DisplayLine[0].TotalWaitingOutput := #TotalWaitingOutputTime;
       #H_CycleMonitor.DisplayLine[0].TotalOutfeedTime := #TotalOutfeedTime;
       #H_CycleMonitor.DisplayLine[0].TotalWaitingEndOfCycle := #TotalWaitingRecoveryTime;
   END_IF;
END_REGION

REGION Network 96: **** 4.4 - Machine Status - Calculated **** Shift display lines one up
   // At EndOfCycle, move all display lines one level up.
   IF #EndOfCyclePulse THEN
       "NotUsedInt" := MOVE_BLK_VARIANT(SRC := #H_CycleMonitor.DisplayLine,
                               COUNT := 10,
                               SRC_INDEX := 0,
                               DEST_INDEX := 0,
                               DEST => #CycleMonitorBuffer.DisplayLine);
       "NotUsedInt" := MOVE_BLK_VARIANT(SRC := #CycleMonitorBuffer.DisplayLine,
                               COUNT := 9,
                               SRC_INDEX := 0,
                               DEST_INDEX := 1,
                               DEST => #H_CycleMonitor.DisplayLine);
   END_IF;
END_REGION

REGION Network 97: **** 4.4 - Machine Status - Calculated **** Reset Time accumulations for new cycle
   // At end of cycle, reset all values
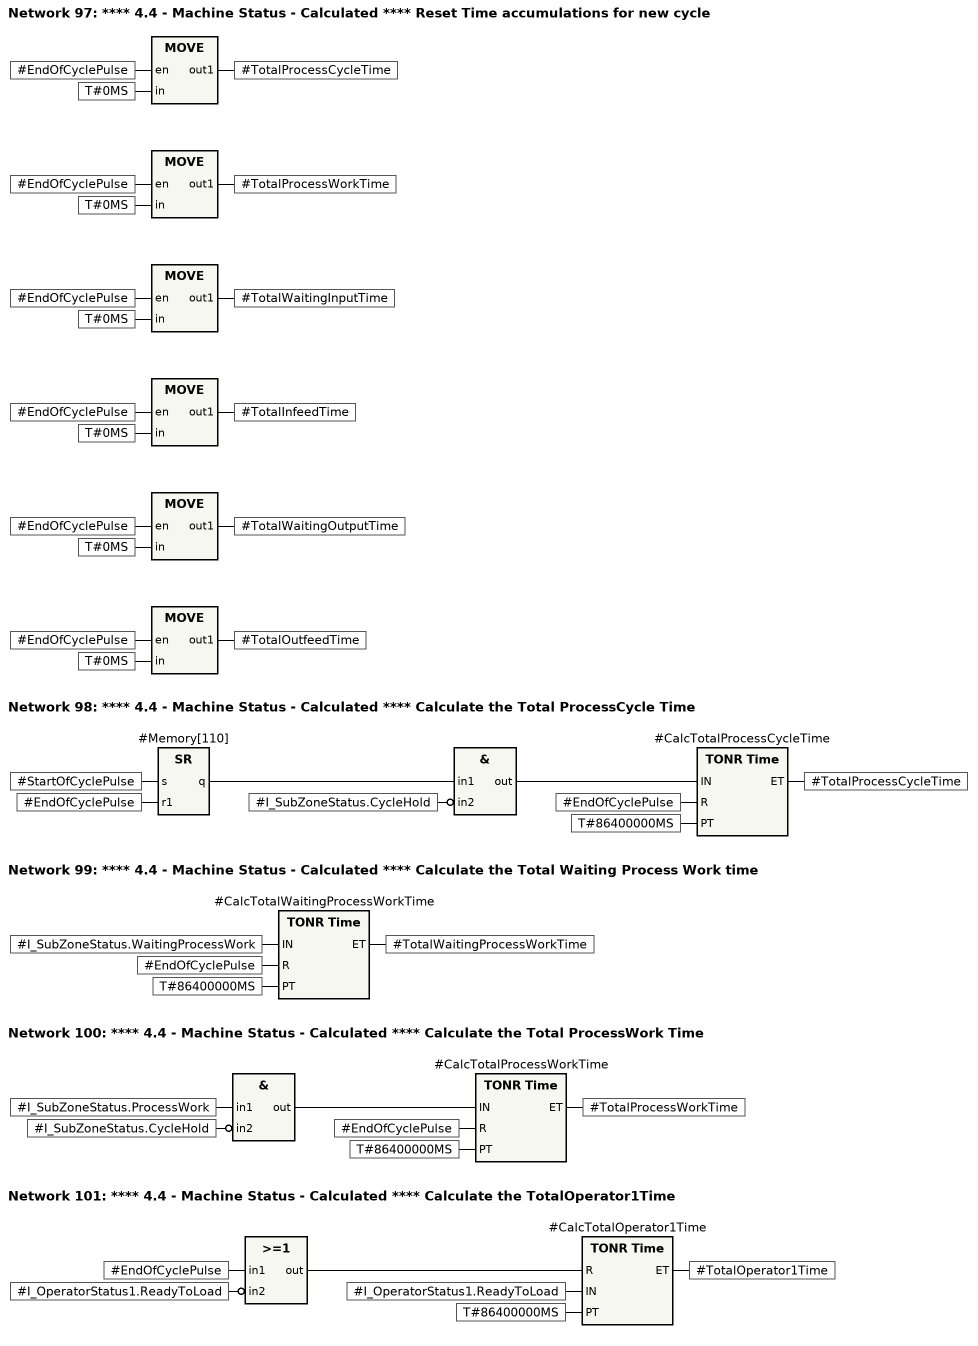
   IF #EndOfCyclePulse THEN
       #TotalProcessCycleTime := T#0MS;
       #TotalProcessWorkTime := T#0MS;
       #TotalWaitingInputTime := T#0MS;
       #TotalInfeedTime := T#0MS;
       #TotalWaitingOutputTime := T#0MS;
       #TotalOutfeedTime := T#0MS;
   END_IF;
END_REGION

REGION Network 98: **** 4.4 - Machine Status - Calculated **** Calculate the Total ProcessCycle Time
   // count local times
   IF #StartOfCyclePulse THEN
       #Memory[110] := TRUE;   // SR flip-flop
   END_IF;
   IF #EndOfCyclePulse THEN #Memory[110] := FALSE; END_IF;
   #CalcTotalProcessCycleTime.TONR(IN := #Memory[110] AND NOT #I_SubZoneStatus.CycleHold,
                           R := #EndOfCyclePulse,
                           PT := T#86400000MS,
                           ET => #TotalProcessCycleTime);
END_REGION

REGION Network 99: **** 4.4 - Machine Status - Calculated **** Calculate the Total Waiting Process Work time
   #CalcTotalWaitingProcessWorkTime.TONR(IN := #I_SubZoneStatus.WaitingProcessWork,
                           R := #EndOfCyclePulse,
                           PT := T#86400000MS,
                           ET => #TotalWaitingProcessWorkTime);
END_REGION

REGION Network 100: **** 4.4 - Machine Status - Calculated **** Calculate the Total ProcessWork Time
   #CalcTotalProcessWorkTime.TONR(IN := #I_SubZoneStatus.ProcessWork AND NOT #I_SubZoneStatus.CycleHold,
                           R := #EndOfCyclePulse,
                           PT := T#86400000MS,
                           ET => #TotalProcessWorkTime);
END_REGION

REGION Network 101: **** 4.4 - Machine Status - Calculated **** Calculate the TotalOperator1Time
   #CalcTotalOperator1Time.TONR(R := #EndOfCyclePulse OR NOT #I_OperatorStatus1.ReadyToLoad,
                           IN := #I_OperatorStatus1.ReadyToLoad,
                           PT := T#86400000MS,
                           ET => #TotalOperator1Time);
END_REGION

REGION Network 102: **** 4.4 - Machine Status - Calculated **** Calculate the TotalOperator2Time
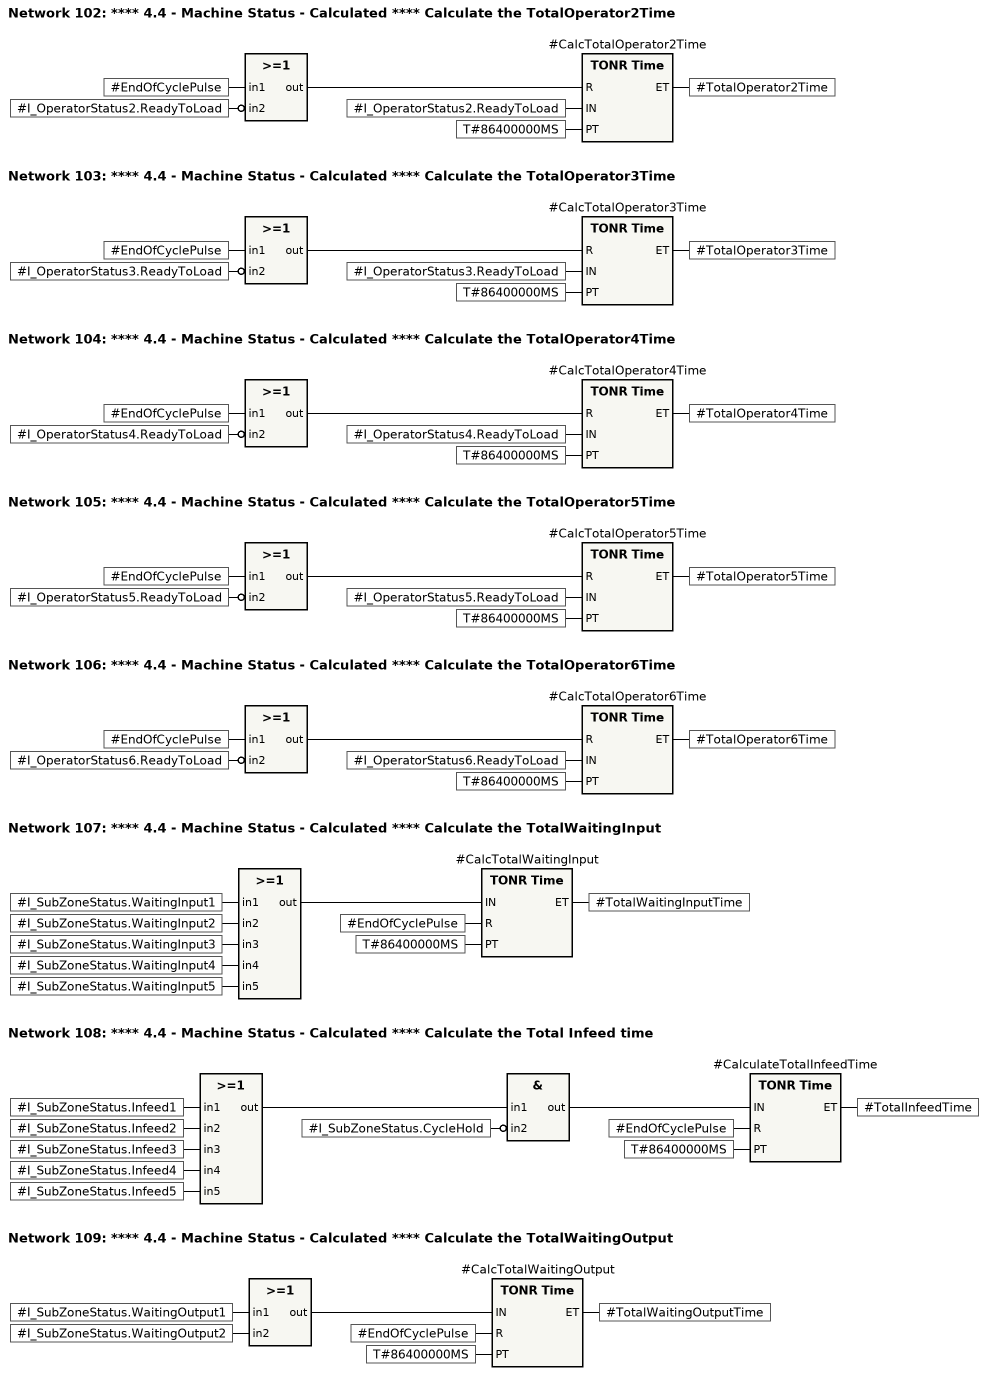
   #CalcTotalOperator2Time.TONR(R := #EndOfCyclePulse OR NOT #I_OperatorStatus2.ReadyToLoad,
                           IN := #I_OperatorStatus2.ReadyToLoad,
                           PT := T#86400000MS,
                           ET => #TotalOperator2Time);
END_REGION

REGION Network 103: **** 4.4 - Machine Status - Calculated **** Calculate the TotalOperator3Time
   #CalcTotalOperator3Time.TONR(R := #EndOfCyclePulse OR NOT #I_OperatorStatus3.ReadyToLoad,
                           IN := #I_OperatorStatus3.ReadyToLoad,
                           PT := T#86400000MS,
                           ET => #TotalOperator3Time);
END_REGION

REGION Network 104: **** 4.4 - Machine Status - Calculated **** Calculate the TotalOperator4Time
   #CalcTotalOperator4Time.TONR(R := #EndOfCyclePulse OR NOT #I_OperatorStatus4.ReadyToLoad,
                           IN := #I_OperatorStatus4.ReadyToLoad,
                           PT := T#86400000MS,
                           ET => #TotalOperator4Time);
END_REGION

REGION Network 105: **** 4.4 - Machine Status - Calculated **** Calculate the TotalOperator5Time
   #CalcTotalOperator5Time.TONR(R := #EndOfCyclePulse OR NOT #I_OperatorStatus5.ReadyToLoad,
                           IN := #I_OperatorStatus5.ReadyToLoad,
                           PT := T#86400000MS,
                           ET => #TotalOperator5Time);
END_REGION

REGION Network 106: **** 4.4 - Machine Status - Calculated **** Calculate the TotalOperator6Time
   #CalcTotalOperator6Time.TONR(R := #EndOfCyclePulse OR NOT #I_OperatorStatus6.ReadyToLoad,
                           IN := #I_OperatorStatus6.ReadyToLoad,
                           PT := T#86400000MS,
                           ET => #TotalOperator6Time);
END_REGION

REGION Network 107: **** 4.4 - Machine Status - Calculated **** Calculate the TotalWaitingInput
   #CalcTotalWaitingInput.TONR(IN := #I_SubZoneStatus.WaitingInput1 OR #I_SubZoneStatus.WaitingInput2 OR #I_SubZoneStatus.WaitingInput3 OR #I_SubZoneStatus.WaitingInput4 OR #I_SubZoneStatus.WaitingInput5,
                           R := #EndOfCyclePulse,
                           PT := T#86400000MS,
                           ET => #TotalWaitingInputTime);
END_REGION

REGION Network 108: **** 4.4 - Machine Status - Calculated **** Calculate the Total Infeed time
   #CalculateTotalInfeedTime(IN := (#I_SubZoneStatus.Infeed1 OR #I_SubZoneStatus.Infeed2 OR #I_SubZoneStatus.Infeed3 OR #I_SubZoneStatus.Infeed4 OR #I_SubZoneStatus.Infeed5) AND NOT #I_SubZoneStatus.CycleHold,   // TONR
                           R := #EndOfCyclePulse,
                           PT := T#86400000MS,
                           ET => #TotalInfeedTime);
END_REGION

REGION Network 109: **** 4.4 - Machine Status - Calculated **** Calculate the TotalWaitingOutput
   #CalcTotalWaitingOutput.TONR(IN := #I_SubZoneStatus.WaitingOutput1 OR #I_SubZoneStatus.WaitingOutput2,
                           R := #EndOfCyclePulse,
                           PT := T#86400000MS,
                           ET => #TotalWaitingOutputTime);
END_REGION

REGION Network 110: **** 4.4 - Machine Status - Calculated **** Calculate the Total Outfeed time
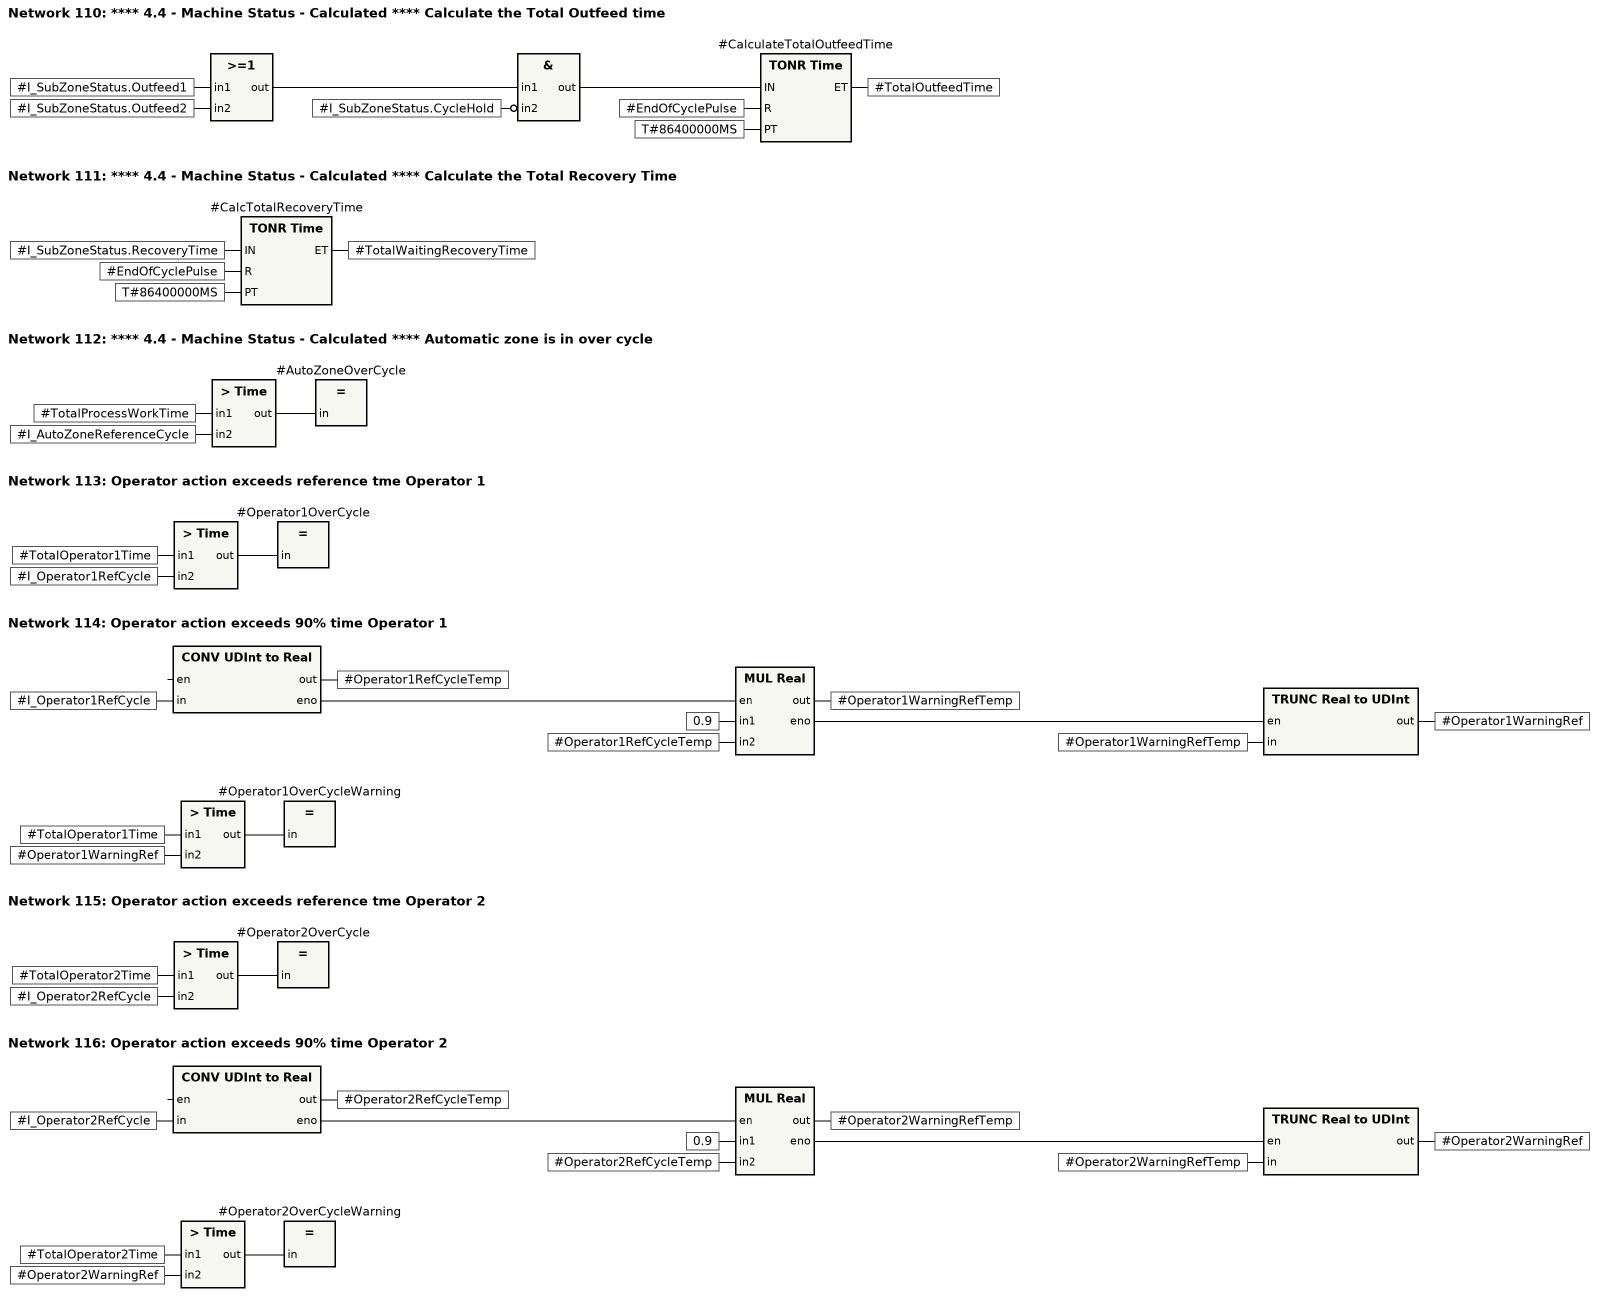
   #CalculateTotalOutfeedTime(IN := (#I_SubZoneStatus.Outfeed1 OR #I_SubZoneStatus.Outfeed2) AND NOT #I_SubZoneStatus.CycleHold,   // TONR
                           R := #EndOfCyclePulse,
                           PT := T#86400000MS,
                           ET => #TotalOutfeedTime);
END_REGION

REGION Network 111: **** 4.4 - Machine Status - Calculated **** Calculate the Total Recovery Time
   #CalcTotalRecoveryTime.TONR(IN := #I_SubZoneStatus.RecoveryTime,
                           R := #EndOfCyclePulse,
                           PT := T#86400000MS,
                           ET => #TotalWaitingRecoveryTime);
END_REGION

REGION Network 112: **** 4.4 - Machine Status - Calculated **** Automatic zone is in over cycle
   // If running time exceeds the auto zone reference time then set the status
   #AutoZoneOverCycle := #TotalProcessWorkTime > #I_AutoZoneReferenceCycle;
END_REGION

REGION Network 113: Operator action exceeds reference tme Operator 1
   #Operator1OverCycle := #TotalOperator1Time > #I_Operator1RefCycle;
END_REGION

REGION Network 114: Operator action exceeds 90% time Operator 1
   #Operator1RefCycleTemp := UDINT_TO_REAL(#I_Operator1RefCycle);
   #Operator1WarningRefTemp := 0.9 * #Operator1RefCycleTemp;
   #Operator1WarningRef := TRUNC(#Operator1WarningRefTemp);
   #Operator1OverCycleWarning := #TotalOperator1Time > #Operator1WarningRef;
END_REGION

REGION Network 115: Operator action exceeds reference tme Operator 2
   #Operator2OverCycle := #TotalOperator2Time > #I_Operator2RefCycle;
END_REGION

REGION Network 116: Operator action exceeds 90% time Operator 2
   #Operator2RefCycleTemp := UDINT_TO_REAL(#I_Operator2RefCycle);
   #Operator2WarningRefTemp := 0.9 * #Operator2RefCycleTemp;
   #Operator2WarningRef := TRUNC(#Operator2WarningRefTemp);
   #Operator2OverCycleWarning := #TotalOperator2Time > #Operator2WarningRef;
END_REGION

REGION Network 117: Operator action exceeds reference tme Operator 3
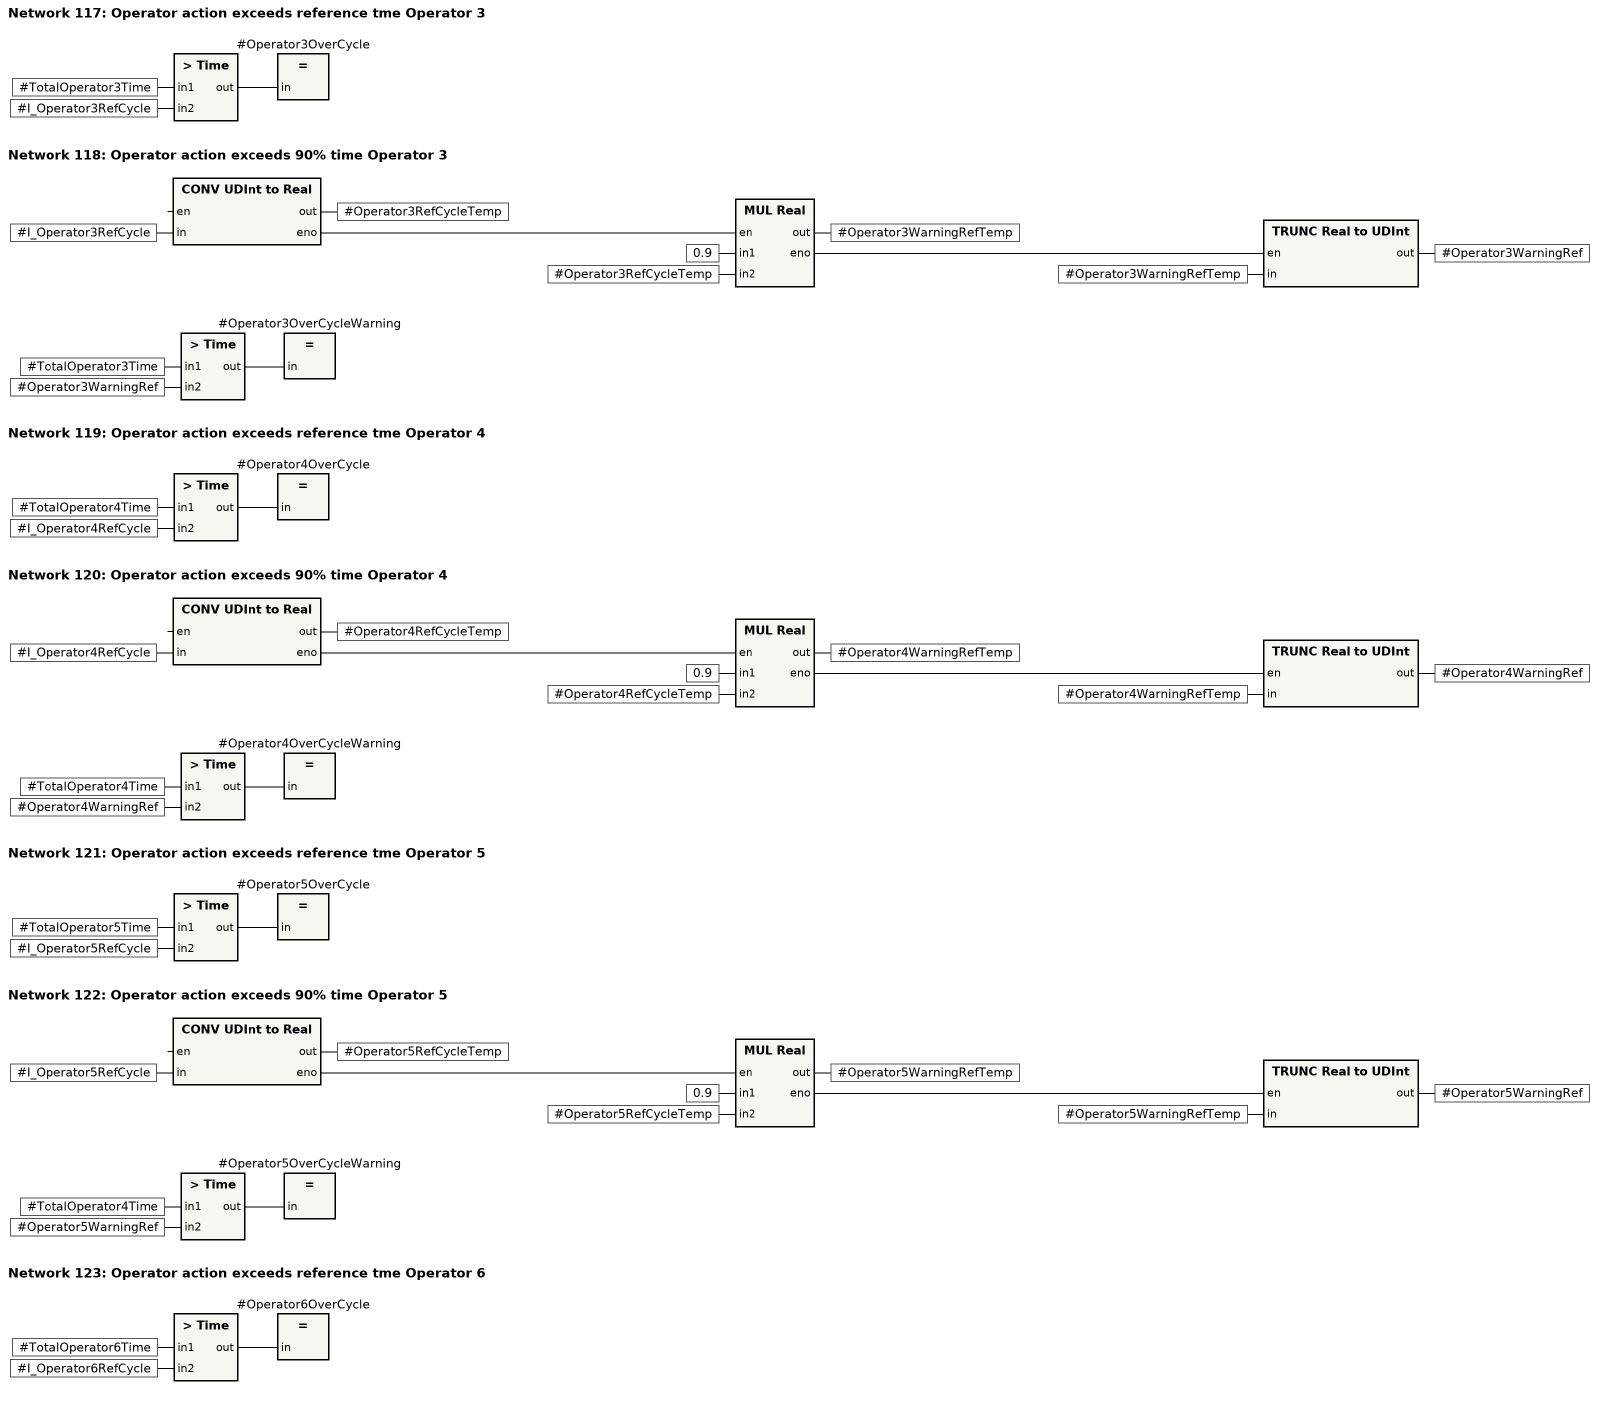
   #Operator3OverCycle := #TotalOperator3Time > #I_Operator3RefCycle;
END_REGION

REGION Network 118: Operator action exceeds 90% time Operator 3
   #Operator3RefCycleTemp := UDINT_TO_REAL(#I_Operator3RefCycle);
   #Operator3WarningRefTemp := 0.9 * #Operator3RefCycleTemp;
   #Operator3WarningRef := TRUNC(#Operator3WarningRefTemp);
   #Operator3OverCycleWarning := #TotalOperator3Time > #Operator3WarningRef;
END_REGION

REGION Network 119: Operator action exceeds reference tme Operator 4
   #Operator4OverCycle := #TotalOperator4Time > #I_Operator4RefCycle;
END_REGION

REGION Network 120: Operator action exceeds 90% time Operator 4
   #Operator4RefCycleTemp := UDINT_TO_REAL(#I_Operator4RefCycle);
   #Operator4WarningRefTemp := 0.9 * #Operator4RefCycleTemp;
   #Operator4WarningRef := TRUNC(#Operator4WarningRefTemp);
   #Operator4OverCycleWarning := #TotalOperator4Time > #Operator4WarningRef;
END_REGION

REGION Network 121: Operator action exceeds reference tme Operator 5
   #Operator5OverCycle := #TotalOperator5Time > #I_Operator5RefCycle;
END_REGION

REGION Network 122: Operator action exceeds 90% time Operator 5
   #Operator5RefCycleTemp := UDINT_TO_REAL(#I_Operator5RefCycle);
   #Operator5WarningRefTemp := 0.9 * #Operator5RefCycleTemp;
   #Operator5WarningRef := TRUNC(#Operator5WarningRefTemp);
   #Operator5OverCycleWarning := #TotalOperator4Time > #Operator5WarningRef;
END_REGION

REGION Network 123: Operator action exceeds reference tme Operator 6
   #Operator6OverCycle := #TotalOperator6Time > #I_Operator6RefCycle;
END_REGION

REGION Network 124: Operator action exceeds 90% time Operator 6
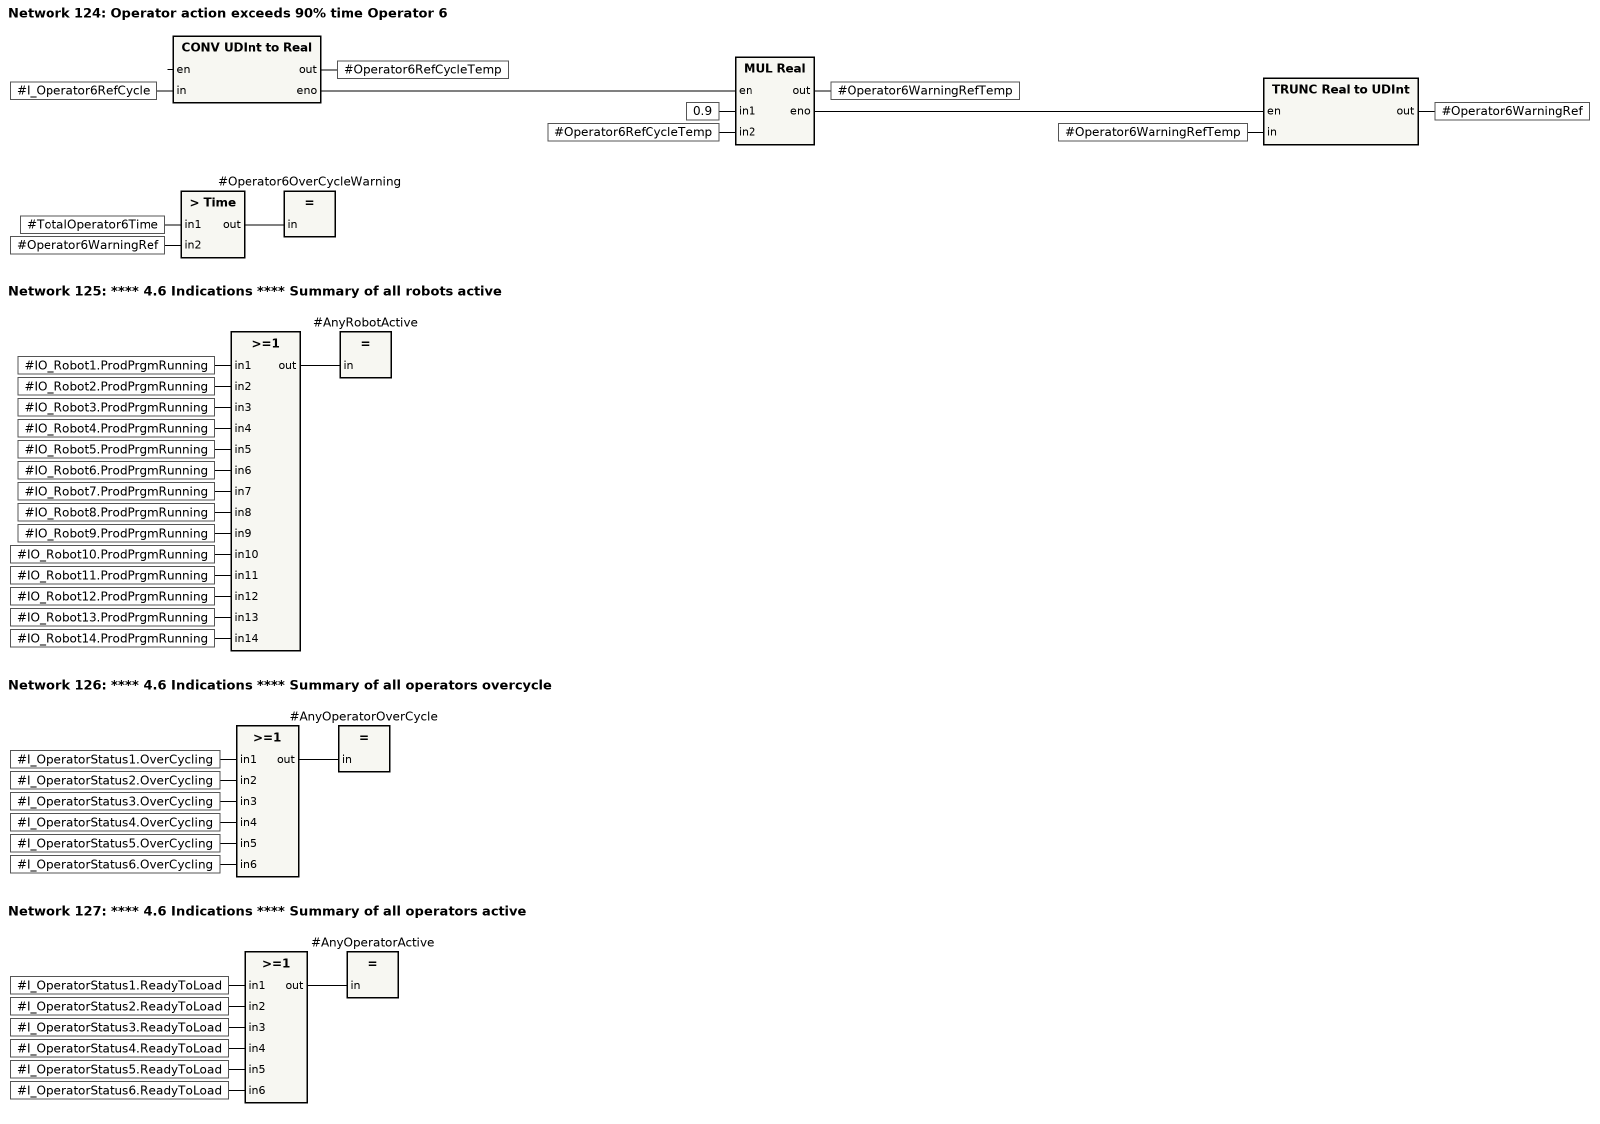
   #Operator6RefCycleTemp := UDINT_TO_REAL(#I_Operator6RefCycle);
   #Operator6WarningRefTemp := 0.9 * #Operator6RefCycleTemp;
   #Operator6WarningRef := TRUNC(#Operator6WarningRefTemp);
   #Operator6OverCycleWarning := #TotalOperator6Time > #Operator6WarningRef;
END_REGION

REGION Network 125: **** 4.6 Indications **** Summary of all robots active
   #AnyRobotActive := #IO_Robot1.ProdPrgmRunning OR #IO_Robot2.ProdPrgmRunning OR #IO_Robot3.ProdPrgmRunning OR #IO_Robot4.ProdPrgmRunning OR #IO_Robot5.ProdPrgmRunning OR #IO_Robot6.ProdPrgmRunning OR #IO_Robot7.ProdPrgmRunning OR #IO_Robot8.ProdPrgmRunning OR #IO_Robot9.ProdPrgmRunning OR #IO_Robot10.ProdPrgmRunning OR #IO_Robot11.ProdPrgmRunning OR #IO_Robot12.ProdPrgmRunning OR #IO_Robot13.ProdPrgmRunning OR #IO_Robot14.ProdPrgmRunning;
END_REGION

REGION Network 126: **** 4.6 Indications **** Summary of all operators overcycle
   #AnyOperatorOverCycle := #I_OperatorStatus1.OverCycling OR #I_OperatorStatus2.OverCycling OR #I_OperatorStatus3.OverCycling OR #I_OperatorStatus4.OverCycling OR #I_OperatorStatus5.OverCycling OR #I_OperatorStatus6.OverCycling;
END_REGION

REGION Network 127: **** 4.6 Indications **** Summary of all operators active
   #AnyOperatorActive := #I_OperatorStatus1.ReadyToLoad OR #I_OperatorStatus2.ReadyToLoad OR #I_OperatorStatus3.ReadyToLoad OR #I_OperatorStatus4.ReadyToLoad OR #I_OperatorStatus5.ReadyToLoad OR #I_OperatorStatus6.ReadyToLoad;
END_REGION

REGION Network 128: **** 4.6 Indications **** Summary of all stopping alarms
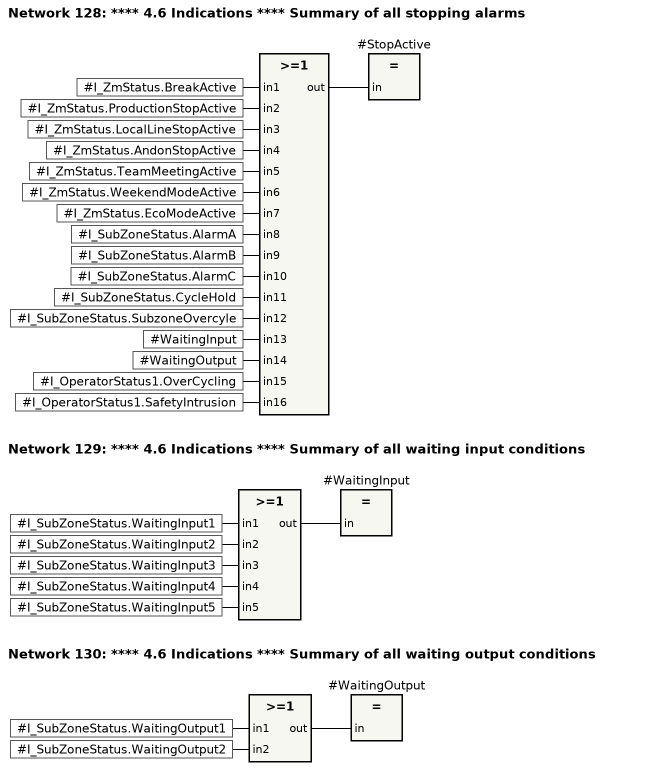
   #StopActive := #I_ZmStatus.BreakActive OR #I_ZmStatus.ProductionStopActive OR #I_ZmStatus.LocalLineStopActive OR #I_ZmStatus.AndonStopActive OR #I_ZmStatus.TeamMeetingActive OR #I_ZmStatus.WeekendModeActive OR #I_ZmStatus.EcoModeActive OR #I_SubZoneStatus.AlarmA OR #I_SubZoneStatus.AlarmB OR #I_SubZoneStatus.AlarmC OR #I_SubZoneStatus.CycleHold OR #I_SubZoneStatus.SubzoneOvercyle OR #WaitingInput OR #WaitingOutput OR #I_OperatorStatus1.OverCycling OR #I_OperatorStatus1.SafetyIntrusion;
END_REGION

REGION Network 129: **** 4.6 Indications **** Summary of all waiting input conditions
   #WaitingInput := #I_SubZoneStatus.WaitingInput1 OR #I_SubZoneStatus.WaitingInput2 OR #I_SubZoneStatus.WaitingInput3 OR #I_SubZoneStatus.WaitingInput4 OR #I_SubZoneStatus.WaitingInput5;
END_REGION

REGION Network 130: **** 4.6 Indications **** Summary of all waiting output conditions
   #WaitingOutput := #I_SubZoneStatus.WaitingOutput1 OR #I_SubZoneStatus.WaitingOutput2;
END_REGION

REGION Network 131: **** 4.6 Indications **** IAnim
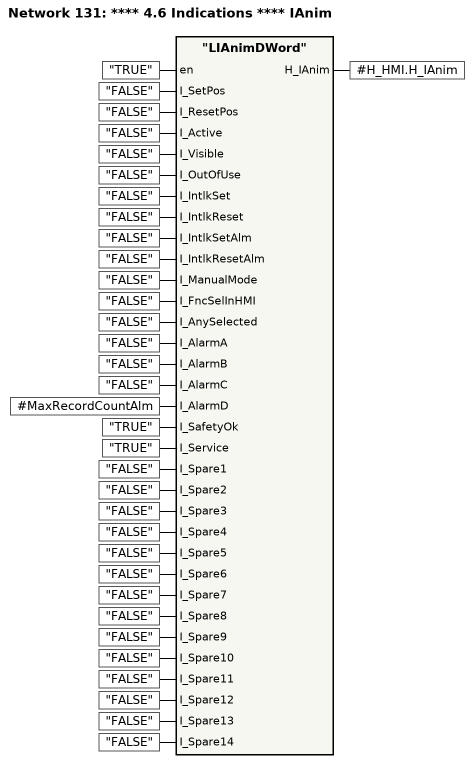
   IF "TRUE" THEN
       "LIAnimDWord"(I_SetPos := "FALSE",
                     I_ResetPos := "FALSE",
                     I_Active := "FALSE",
                     I_Visible := "FALSE",
                     I_OutOfUse := "FALSE",
                     I_IntlkSet := "FALSE",
                     I_IntlkReset := "FALSE",
                     I_IntlkSetAlm := "FALSE",
                     I_IntlkResetAlm := "FALSE",
                     I_ManualMode := "FALSE",
                     I_FncSelInHMI := "FALSE",
                     I_AnySelected := "FALSE",
                     I_AlarmA := "FALSE",
                     I_AlarmB := "FALSE",
                     I_AlarmC := "FALSE",
                     I_AlarmD := #MaxRecordCountAlm,
                     I_SafetyOk := "TRUE",
                     I_Service := "TRUE",
                     I_Spare1 := "FALSE",
                     I_Spare2 := "FALSE",
                     I_Spare3 := "FALSE",
                     I_Spare4 := "FALSE",
                     I_Spare5 := "FALSE",
                     I_Spare6 := "FALSE",
                     I_Spare7 := "FALSE",
                     I_Spare8 := "FALSE",
                     I_Spare9 := "FALSE",
                     I_Spare10 := "FALSE",
                     I_Spare11 := "FALSE",
                     I_Spare12 := "FALSE",
                     I_Spare13 := "FALSE",
                     I_Spare14 := "FALSE",
                     H_IAnim => #H_HMI.H_IAnim);
   END_IF;
END_REGION

REGION Network 132: **** 4.6 Indications **** AnimW1
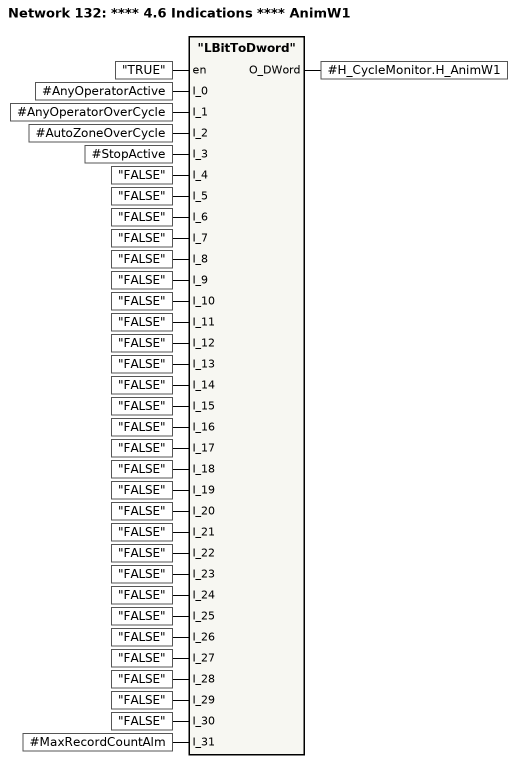
   IF "TRUE" THEN
       "LBitToDword"(I_0 := #AnyOperatorActive,
                     I_1 := #AnyOperatorOverCycle,
                     I_2 := #AutoZoneOverCycle,
                     I_3 := #StopActive,
                     I_4 := "FALSE",
                     I_5 := "FALSE",
                     I_6 := "FALSE",
                     I_7 := "FALSE",
                     I_8 := "FALSE",
                     I_9 := "FALSE",
                     I_10 := "FALSE",
                     I_11 := "FALSE",
                     I_12 := "FALSE",
                     I_13 := "FALSE",
                     I_14 := "FALSE",
                     I_15 := "FALSE",
                     I_16 := "FALSE",
                     I_17 := "FALSE",
                     I_18 := "FALSE",
                     I_19 := "FALSE",
                     I_20 := "FALSE",
                     I_21 := "FALSE",
                     I_22 := "FALSE",
                     I_23 := "FALSE",
                     I_24 := "FALSE",
                     I_25 := "FALSE",
                     I_26 := "FALSE",
                     I_27 := "FALSE",
                     I_28 := "FALSE",
                     I_29 := "FALSE",
                     I_30 := "FALSE",
                     I_31 := #MaxRecordCountAlm,
                     O_DWord => #H_CycleMonitor.H_AnimW1);
   END_IF;
END_REGION

REGION Network 133: **** 4.6 Indications **** AnimW2
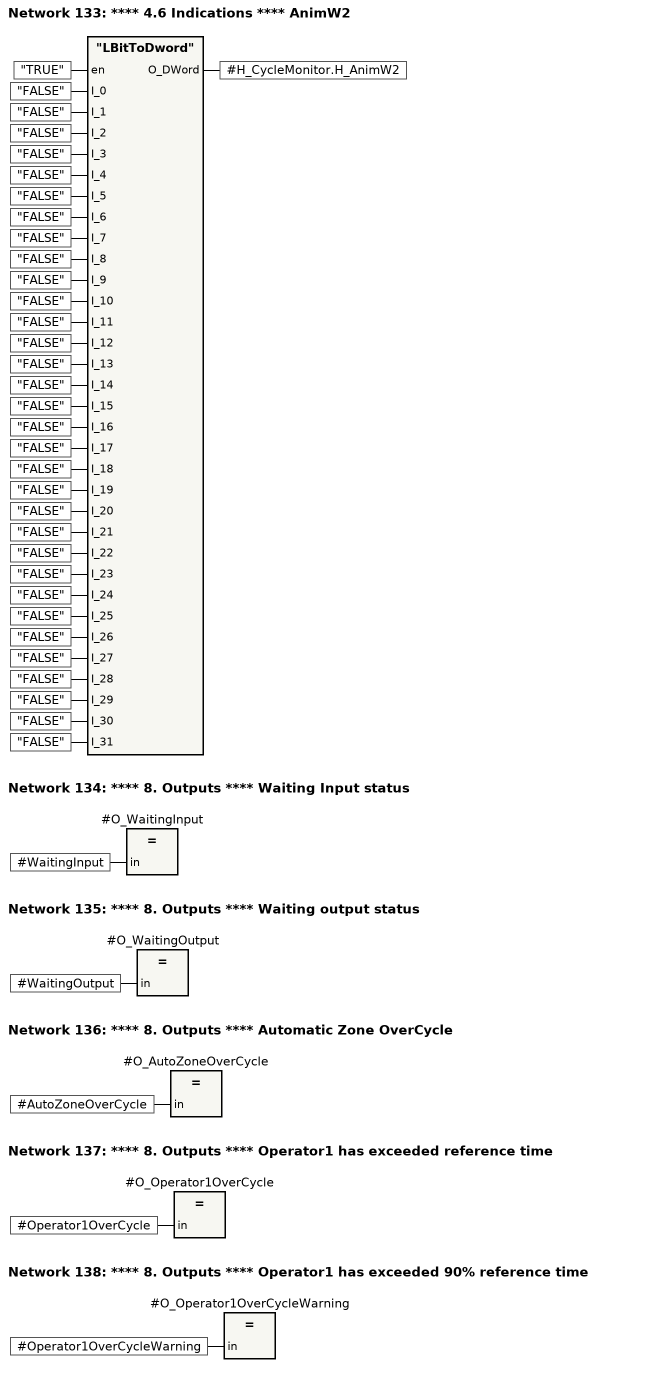
   IF "TRUE" THEN
       "LBitToDword"(I_0 := "FALSE",
                     I_1 := "FALSE",
                     I_2 := "FALSE",
                     I_3 := "FALSE",
                     I_4 := "FALSE",
                     I_5 := "FALSE",
                     I_6 := "FALSE",
                     I_7 := "FALSE",
                     I_8 := "FALSE",
                     I_9 := "FALSE",
                     I_10 := "FALSE",
                     I_11 := "FALSE",
                     I_12 := "FALSE",
                     I_13 := "FALSE",
                     I_14 := "FALSE",
                     I_15 := "FALSE",
                     I_16 := "FALSE",
                     I_17 := "FALSE",
                     I_18 := "FALSE",
                     I_19 := "FALSE",
                     I_20 := "FALSE",
                     I_21 := "FALSE",
                     I_22 := "FALSE",
                     I_23 := "FALSE",
                     I_24 := "FALSE",
                     I_25 := "FALSE",
                     I_26 := "FALSE",
                     I_27 := "FALSE",
                     I_28 := "FALSE",
                     I_29 := "FALSE",
                     I_30 := "FALSE",
                     I_31 := "FALSE",
                     O_DWord => #H_CycleMonitor.H_AnimW2);
   END_IF;
END_REGION

REGION Network 134: **** 8. Outputs **** Waiting Input status
   #O_WaitingInput := #WaitingInput;
END_REGION

REGION Network 135: **** 8. Outputs **** Waiting output status
   #O_WaitingOutput := #WaitingOutput;
END_REGION

REGION Network 136: **** 8. Outputs **** Automatic Zone OverCycle
   #O_AutoZoneOverCycle := #AutoZoneOverCycle;
END_REGION

REGION Network 137: **** 8. Outputs **** Operator1 has exceeded reference time
   #O_Operator1OverCycle := #Operator1OverCycle;
END_REGION

REGION Network 138: **** 8. Outputs **** Operator1 has exceeded 90% reference time
   #O_Operator1OverCycleWarning := #Operator1OverCycleWarning;
END_REGION

REGION Network 139: **** 8. Outputs **** Operator2 has exceeded reference time
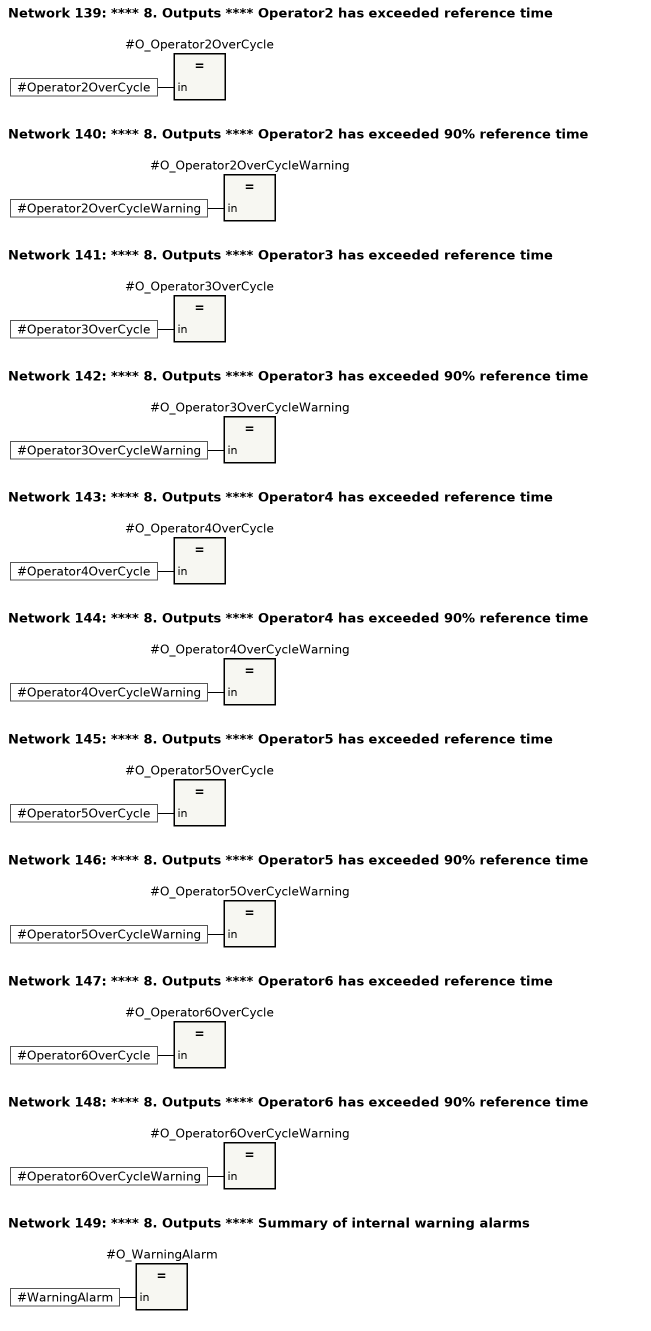
   #O_Operator2OverCycle := #Operator2OverCycle;
END_REGION

REGION Network 140: **** 8. Outputs **** Operator2 has exceeded 90% reference time
   #O_Operator2OverCycleWarning := #Operator2OverCycleWarning;
END_REGION

REGION Network 141: **** 8. Outputs **** Operator3 has exceeded reference time
   #O_Operator3OverCycle := #Operator3OverCycle;
END_REGION

REGION Network 142: **** 8. Outputs **** Operator3 has exceeded 90% reference time
   #O_Operator3OverCycleWarning := #Operator3OverCycleWarning;
END_REGION

REGION Network 143: **** 8. Outputs **** Operator4 has exceeded reference time
   #O_Operator4OverCycle := #Operator4OverCycle;
END_REGION

REGION Network 144: **** 8. Outputs **** Operator4 has exceeded 90% reference time
   #O_Operator4OverCycleWarning := #Operator4OverCycleWarning;
END_REGION

REGION Network 145: **** 8. Outputs **** Operator5 has exceeded reference time
   #O_Operator5OverCycle := #Operator5OverCycle;
END_REGION

REGION Network 146: **** 8. Outputs **** Operator5 has exceeded 90% reference time
   #O_Operator5OverCycleWarning := #Operator5OverCycleWarning;
END_REGION

REGION Network 147: **** 8. Outputs **** Operator6 has exceeded reference time
   #O_Operator6OverCycle := #Operator6OverCycle;
END_REGION

REGION Network 148: **** 8. Outputs **** Operator6 has exceeded 90% reference time
   #O_Operator6OverCycleWarning := #Operator6OverCycleWarning;
END_REGION

REGION Network 149: **** 8. Outputs **** Summary of internal warning alarms
   #O_WarningAlarm := #WarningAlarm;
END_REGION
END_FUNCTION_BLOCK
